LIN {X 0,Y 227.847,Z 291.73,A -85,B 0,C 180,E1 -20016.68,E2 -20016.68} C_VEL
LIN {X 0,Y 227.819,Z 291.734,A -85,B 0,C 180,E1 -20020.379,E2 -20020.379} C_VEL
LIN {X 0,Y 227.828,Z 291.733,A -85,B 0,C 180,E1 -20025.195,E2 -20025.195} C_VEL
LIN {X 0,Y 227.828,Z 291.729,A -85,B 0,C 180,E1 -20029.623,E2 -20029.623} C_VEL
LIN {X 0,Y 227.883,Z 291.723,A -85,B 0,C 180,E1 -20034.128,E2 -20034.128} C_VEL
LIN {X 0,Y 227.87,Z 291.726,A -85,B 0,C 180,E1 -20038.377,E2 -20038.377} C_VEL
LIN {X 0,Y 227.882,Z 291.725,A -85,B 0,C 180,E1 -20042.444,E2 -20042.444} C_VEL
LIN {X 0,Y 227.916,Z 291.719,A -85,B 0,C 180,E1 -20046.368,E2 -20046.368} C_VEL
LIN {X 0,Y 227.945,Z 291.716,A -85,B 0,C 180,E1 -20050.175,E2 -20050.175} C_VEL
LIN {X 0,Y 228.061,Z 291.7,A -85,B 0,C 180,E1 -20053.898,E2 -20053.898} C_VEL
LIN {X 0,Y 228.076,Z 291.698,A -85,B 0,C 180,E1 -20057.543,E2 -20057.543} C_VEL
LIN {X 0,Y 228.26,Z 291.674,A -85,B 0,C 180,E1 -20061.144,E2 -20061.144} C_VEL
LIN {X 0,Y 228.31,Z 291.666,A -85,B 0,C 180,E1 -20062.927,E2 -20062.927} C_VEL
LIN {X 0,Y 228.552,Z 291.64,A -85,B 0,C 180,E1 -20068.238,E2 -20068.238} C_VEL
LIN {X 0,Y 228.554,Z 291.638,A -85,B 0,C 180,E1 -20071.762,E2 -20071.762} C_VEL
LIN {X 0,Y 228.313,Z 291.668,A -85,B 0,C 180,E1 -20077.073,E2 -20077.073} C_VEL
LIN {X 0,Y 228.149,Z 291.687,A -85,B 0,C 180,E1 -20080.651,E2 -20080.651} C_VEL
LIN {X 0,Y 228.068,Z 291.699,A -85,B 0,C 180,E1 -20084.272,E2 -20084.272} C_VEL
LIN {X 0,Y 228.01,Z 291.706,A -85,B 0,C 180,E1 -20087.953,E2 -20087.953} C_VEL
LIN {X 0,Y 227.964,Z 291.712,A -85,B 0,C 180,E1 -20092.348,E2 -20092.348} C_VEL
LIN {X 0,Y 227.945,Z 291.712,A -85,B 0,C 180,E1 -20096.602,E2 -20096.602} C_VEL
LIN {X 0,Y 227.9,Z 291.72,A -85,B 0,C 180,E1 -20100.291,E2 -20100.291} C_VEL
LIN {X 0,Y 227.879,Z 291.72,A -85,B 0,C 180,E1 -20103.72,E2 -20103.72} C_VEL
LIN {X 0,Y 227.842,Z 291.727,A -85,B 0,C 180,E1 -20108.092,E2 -20108.092} C_VEL
LIN {X 0,Y 227.794,Z 291.733,A -85,B 0,C 180,E1 -20112.747,E2 -20112.747} C_VEL
LIN {X 0,Y 227.808,Z 291.733,A -85,B 0,C 180,E1 -20117.256,E2 -20117.256} C_VEL
LIN {X 0,Y 227.847,Z 291.725,A -85,B 0,C 180,E1 -20121.909,E2 -20121.909} C_VEL
LIN {X 0,Y 227.882,Z 291.724,A -85,B 0,C 180,E1 -20126.377,E2 -20126.377} C_VEL
LIN {X 0,Y 227.908,Z 291.719,A -85,B 0,C 180,E1 -20130.436,E2 -20130.436} C_VEL
LIN {X 0,Y 227.932,Z 291.719,A -85,B 0,C 180,E1 -20134.426,E2 -20134.426} C_VEL
LIN {X 0,Y 227.965,Z 291.712,A -85,B 0,C 180,E1 -20138.287,E2 -20138.287} C_VEL
LIN {X 0,Y 228.038,Z 291.703,A -85,B 0,C 180,E1 -20142.825,E2 -20142.825} C_VEL
LIN {X 0,Y 228.076,Z 291.697,A -85,B 0,C 180,E1 -20147.543,E2 -20147.543} C_VEL
LIN {X 0,Y 228.261,Z 291.674,A -85,B 0,C 180,E1 -20151.144,E2 -20151.144} C_VEL
LIN {X 0,Y 228.31,Z 291.666,A -85,B 0,C 180,E1 -20152.927,E2 -20152.927} C_VEL
LIN {X 0,Y 228.554,Z 291.641,A -85,B 0,C 180,E1 -20158.237,E2 -20158.237} C_VEL
LIN {X 0,Y 228.555,Z 291.639,A -85,B 0,C 180,E1 -20161.762,E2 -20161.762} C_VEL
LIN {X 0,Y 228.311,Z 291.669,A -85,B 0,C 180,E1 -20167.072,E2 -20167.072} C_VEL
LIN {X 0,Y 228.148,Z 291.687,A -85,B 0,C 180,E1 -20170.651,E2 -20170.651} C_VEL
LIN {X 0,Y 228.067,Z 291.7,A -85,B 0,C 180,E1 -20174.271,E2 -20174.271} C_VEL
LIN {X 0,Y 228.006,Z 291.706,A -85,B 0,C 180,E1 -20177.953,E2 -20177.953} C_VEL
LIN {X 0,Y 227.925,Z 291.718,A -85,B 0,C 180,E1 -20182.324,E2 -20182.324} C_VEL
LIN {X 0,Y 227.949,Z 291.73,A -85,B 0,C 180,E1 -20185.571,E2 -20185.571} C_VEL
LIN {X 0,Y 228.569,Z 295.999,A -85,B 0,C 180,E1 -20190.577,E2 -20190.577} C_VEL
LIN {X 0,Y 229.068,Z 299.133,A -85,B 0,C 180,E1 -20194.066,E2 -20194.066} C_VEL
LIN {X 0,Y 229.908,Z 303.616,A -85,B 0,C 180,E1 -20198.804,E2 -20198.804} C_VEL
LIN {X 0,Y 230.865,Z 307.87,A -85,B 0,C 180,E1 -20203.062,E2 -20203.062} C_VEL
LIN {X 0,Y 231.268,Z 310.585,A -85,B 0,C 180,E1 -20205.657,E2 -20205.657} C_VEL
LIN {X 0,Y 231.214,Z 313.163,A -85,B 0,C 180,E1 -20208.032,E2 -20208.032} C_VEL
LIN {X 0,Y 230.92,Z 314.73,A -85,B 0,C 180,E1 -20209.433,E2 -20209.433} C_VEL
LIN {X 0,Y 234.651,Z 334.28,A -85,B 0,C 180,E1 -20211.37,E2 -20211.37} C_VEL
LIN {X 0,Y 237.634,Z 350.876,A -85,B 0,C 180,E1 -20213.342,E2 -20213.342} C_VEL
LIN {X 0,Y 240.205,Z 366.69,A -85,B 0,C 180,E1 -20215.507,E2 -20215.507} C_VEL
LIN {X 0,Y 240.445,Z 368.284,A -85,B 0,C 180,E1 -20215.742,E2 -20215.742} C_VEL
LIN {X 0,Y 240.526,Z 373.392,A -85,B 0,C 180,E1 -20216.468,E2 -20216.468} C_VEL
LIN {X 0,Y 239.415,Z 378.527,A -85,B 0,C 180,E1 -20217.164,E2 -20217.164} C_VEL
LIN {X 0,Y 235.584,Z 388.411,A -85,B 0,C 180,E1 -20218.588,E2 -20218.588} C_VEL
LIN {X 0,Y 233.418,Z 394.85,A -85,B 0,C 180,E1 -20219.67,E2 -20219.67} C_VEL
LIN {X 0,Y 230.045,Z 407.856,A -85,B 0,C 180,E1 -20222.281,E2 -20222.281} C_VEL
LIN {X 0,Y 227.246,Z 418.384,A -85,B 0,C 180,E1 -20224.834,E2 -20224.834} C_VEL
LIN {X 0,Y 224.584,Z 429.031,A -85,B 0,C 180,E1 -20227.943,E2 -20227.943} C_VEL
LIN {X 0,Y 222.201,Z 439.134,A -85,B 0,C 180,E1 -20231.561,E2 -20231.561} C_VEL
LIN {X 0,Y 220.517,Z 447.367,A -85,B 0,C 180,E1 -20235.228,E2 -20235.228} C_VEL
LIN {X 0,Y 219.526,Z 453.947,A -85,B 0,C 180,E1 -20238.925,E2 -20238.925} C_VEL
LIN {X 0,Y 219.139,Z 459.038,A -85,B 0,C 180,E1 -20242.629,E2 -20242.629} C_VEL
LIN {X 0,Y 219.1,Z 461.063,A -85,B 0,C 180,E1 -20244.478,E2 -20244.478} C_VEL
LIN {X 0,Y 218.927,Z 464.073,A -85,B 0,C 180,E1 -20248.16,E2 -20248.16} C_VEL
LIN {X 0,Y 218.978,Z 465.12,A -85,B 0,C 180,E1 -20250,E2 -20250} C_VEL
LIN {X 0,Y 218.835,Z 466.296,A -85,B 0,C 180,E1 -20253.683,E2 -20253.683} C_VEL
LIN {X 0,Y 218.754,Z 466.325,A -85,B 0,C 180,E1 -20257.383,E2 -20257.383} C_VEL
LIN {X 0,Y 219.17,Z 465.303,A -85,B 0,C 180,E1 -20261.093,E2 -20261.093} C_VEL
LIN {X 0,Y 220.392,Z 463.369,A -85,B 0,C 180,E1 -20264.78,E2 -20264.78} C_VEL
LIN {X 0,Y 222.497,Z 460.267,A -85,B 0,C 180,E1 -20268.63,E2 -20268.63} C_VEL
LIN {X 0,Y 227.181,Z 454.516,A -85,B 0,C 180,E1 -20273.714,E2 -20273.714} C_VEL
LIN {X 0,Y 232.726,Z 448.077,A -85,B 0,C 180,E1 -20277.91,E2 -20277.91} C_VEL
LIN {X 0,Y 238.908,Z 441.296,A -85,B 0,C 180,E1 -20281.385,E2 -20281.385} C_VEL
LIN {X 0,Y 246.615,Z 433.163,A -85,B 0,C 180,E1 -20284.747,E2 -20284.747} C_VEL
LIN {X 0,Y 256.413,Z 423.002,A -85,B 0,C 180,E1 -20288.076,E2 -20288.076} C_VEL
LIN {X 0,Y 266.397,Z 412.614,A -85,B 0,C 180,E1 -20290.764,E2 -20290.764} C_VEL
LIN {X 0,Y 269.564,Z 409.165,A -85,B 0,C 180,E1 -20291.67,E2 -20291.67} C_VEL
LIN {X 0,Y 273.733,Z 404.367,A -85,B 0,C 180,E1 -20293.189,E2 -20293.189} C_VEL
LIN {X 0,Y 276.225,Z 401.494,A -85,B 0,C 180,E1 -20294.569,E2 -20294.569} C_VEL
LIN {X 0,Y 276.98,Z 400.651,A -85,B 0,C 180,E1 -20295.273,E2 -20295.273} C_VEL
LIN {X 0,Y 276.699,Z 400.883,A -85,B 0,C 180,E1 -20295.995,E2 -20295.995} C_VEL
LIN {X 0,Y 265.948,Z 410.924,A -85,B 0,C 180,E1 -20298.651,E2 -20298.651} C_VEL
LIN {X 0,Y 255.652,Z 420.112,A -85,B 0,C 180,E1 -20301.791,E2 -20301.791} C_VEL
LIN {X 0,Y 246.651,Z 427.81,A -85,B 0,C 180,E1 -20305.259,E2 -20305.259} C_VEL
LIN {X 0,Y 238.941,Z 434.054,A -85,B 0,C 180,E1 -20309.021,E2 -20309.021} C_VEL
LIN {X 0,Y 232.51,Z 438.799,A -85,B 0,C 180,E1 -20313.038,E2 -20313.038} C_VEL
LIN {X 0,Y 228.346,Z 441.537,A -85,B 0,C 180,E1 -20316.415,E2 -20316.415} C_VEL
LIN {X 0,Y 224.998,Z 443.249,A -85,B 0,C 180,E1 -20319.904,E2 -20319.904} C_VEL
LIN {X 0,Y 222.398,Z 443.986,A -85,B 0,C 180,E1 -20323.477,E2 -20323.477} C_VEL
LIN {X 0,Y 220.643,Z 443.701,A -85,B 0,C 180,E1 -20327.117,E2 -20327.117} C_VEL
LIN {X 0,Y 219.572,Z 442.329,A -85,B 0,C 180,E1 -20330.791,E2 -20330.791} C_VEL
LIN {X 0,Y 219.064,Z 439.811,A -85,B 0,C 180,E1 -20334.477,E2 -20334.477} C_VEL
LIN {X 0,Y 218.944,Z 436.124,A -85,B 0,C 180,E1 -20338.161,E2 -20338.161} C_VEL
LIN {X 0,Y 219.045,Z 431.191,A -85,B 0,C 180,E1 -20341.839,E2 -20341.839} C_VEL
LIN {X 0,Y 219.67,Z 424.882,A -85,B 0,C 180,E1 -20345.508,E2 -20345.508} C_VEL
LIN {X 0,Y 220.495,Z 417.013,A -85,B 0,C 180,E1 -20349.171,E2 -20349.171} C_VEL
LIN {X 0,Y 221.966,Z 407.428,A -85,B 0,C 180,E1 -20352.806,E2 -20352.806} C_VEL
LIN {X 0,Y 223.778,Z 397.372,A -85,B 0,C 180,E1 -20355.951,E2 -20355.951} C_VEL
LIN {X 0,Y 226.003,Z 385.408,A -85,B 0,C 180,E1 -20359.058,E2 -20359.058} C_VEL
LIN {X 0,Y 228.56,Z 372.174,A -85,B 0,C 180,E1 -20361.891,E2 -20361.891} C_VEL
LIN {X 0,Y 231.022,Z 358.568,A -85,B 0,C 180,E1 -20364.316,E2 -20364.316} C_VEL
LIN {X 0,Y 233.545,Z 344.768,A -85,B 0,C 180,E1 -20366.351,E2 -20366.351} C_VEL
LIN {X 0,Y 234.092,Z 341.635,A -85,B 0,C 180,E1 -20366.766,E2 -20366.766} C_VEL
LIN {X 0,Y 233.603,Z 337.571,A -85,B 0,C 180,E1 -20367.358,E2 -20367.358} C_VEL
LIN {X 0,Y 230.249,Z 323.156,A -85,B 0,C 180,E1 -20369.415,E2 -20369.415} C_VEL
LIN {X 0,Y 227.217,Z 312.166,A -85,B 0,C 180,E1 -20370.87,E2 -20370.87} C_VEL
LIN {X 0,Y 221.231,Z 294.789,A -85,B 0,C 180,E1 -20373.004,E2 -20373.004} C_VEL
LIN {X 0,Y 220.601,Z 292.633,A -85,B 0,C 180,E1 -20373.269,E2 -20373.269} C_VEL
LIN {X 0,Y 220.793,Z 292.611,A -85,B 0,C 180,E1 -20377.272,E2 -20377.272} C_VEL
LIN {X 0,Y 220.769,Z 292.612,A -85,B 0,C 180,E1 -20381.954,E2 -20381.954} C_VEL
LIN {X 0,Y 220.77,Z 292.61,A -85,B 0,C 180,E1 -20385.545,E2 -20385.545} C_VEL
LIN {X 0,Y 220.809,Z 292.605,A -85,B 0,C 180,E1 -20390.463,E2 -20390.463} C_VEL
LIN {X 0,Y 220.803,Z 292.606,A -85,B 0,C 180,E1 -20395.045,E2 -20395.045} C_VEL
LIN {X 0,Y 220.837,Z 292.6,A -85,B 0,C 180,E1 -20399.39,E2 -20399.39} C_VEL
LIN {X 0,Y 220.897,Z 292.592,A -85,B 0,C 180,E1 -20403.55,E2 -20403.55} C_VEL
LIN {X 0,Y 220.88,Z 292.592,A -85,B 0,C 180,E1 -20407.554,E2 -20407.554} C_VEL
LIN {X 0,Y 220.987,Z 292.582,A -85,B 0,C 180,E1 -20412.571,E2 -20412.571} C_VEL
LIN {X 0,Y 221.015,Z 292.577,A -85,B 0,C 180,E1 -20417.139,E2 -20417.139} C_VEL
LIN {X 0,Y 221.2,Z 292.554,A -85,B 0,C 180,E1 -20420.859,E2 -20420.859} C_VEL
LIN {X 0,Y 221.247,Z 292.546,A -85,B 0,C 180,E1 -20422.7,E2 -20422.7} C_VEL
LIN {X 0,Y 221.509,Z 292.518,A -85,B 0,C 180,E1 -20428.182,E2 -20428.182} C_VEL
LIN {X 0,Y 221.512,Z 292.516,A -85,B 0,C 180,E1 -20431.818,E2 -20431.818} C_VEL
LIN {X 0,Y 221.25,Z 292.549,A -85,B 0,C 180,E1 -20437.3,E2 -20437.3} C_VEL
LIN {X 0,Y 221.07,Z 292.569,A -85,B 0,C 180,E1 -20440.996,E2 -20440.996} C_VEL
LIN {X 0,Y 220.999,Z 292.579,A -85,B 0,C 180,E1 -20444.739,E2 -20444.739} C_VEL
LIN {X 0,Y 220.931,Z 292.586,A -85,B 0,C 180,E1 -20448.549,E2 -20448.549} C_VEL
LIN {X 0,Y 220.924,Z 292.589,A -85,B 0,C 180,E1 -20452.698,E2 -20452.698} C_VEL
LIN {X 0,Y 220.887,Z 292.592,A -85,B 0,C 180,E1 -20457.014,E2 -20457.014} C_VEL
LIN {X 0,Y 220.841,Z 292.6,A -85,B 0,C 180,E1 -20460.768,E2 -20460.768} C_VEL
LIN {X 0,Y 220.796,Z 292.604,A -85,B 0,C 180,E1 -20464.956,E2 -20464.956} C_VEL
LIN {X 0,Y 220.804,Z 292.607,A -85,B 0,C 180,E1 -20467.275,E2 -20467.275} C_VEL
LIN {X 0,Y 220.754,Z 292.607,A -85,B 0,C 180,E1 -20471.957,E2 -20471.957} C_VEL
LIN {X 0,Y 220.768,Z 292.609,A -85,B 0,C 180,E1 -20475.544,E2 -20475.544} C_VEL
LIN {X 0,Y 220.809,Z 292.602,A -85,B 0,C 180,E1 -20480.463,E2 -20480.463} C_VEL
LIN {X 0,Y 220.804,Z 292.606,A -85,B 0,C 180,E1 -20485.045,E2 -20485.045} C_VEL
LIN {X 0,Y 220.837,Z 292.598,A -85,B 0,C 180,E1 -20489.39,E2 -20489.39} C_VEL
LIN {X 0,Y 220.898,Z 292.592,A -85,B 0,C 180,E1 -20493.549,E2 -20493.549} C_VEL
LIN {X 0,Y 220.881,Z 292.591,A -85,B 0,C 180,E1 -20497.553,E2 -20497.553} C_VEL
LIN {X 0,Y 220.988,Z 292.583,A -85,B 0,C 180,E1 -20502.571,E2 -20502.571} C_VEL
LIN {X 0,Y 221.015,Z 292.577,A -85,B 0,C 180,E1 -20507.138,E2 -20507.138} C_VEL
LIN {X 0,Y 221.2,Z 292.554,A -85,B 0,C 180,E1 -20510.859,E2 -20510.859} C_VEL
LIN {X 0,Y 221.126,Z 292.564,A -85,B 0,C 180,E1 -20514.528,E2 -20514.528} C_VEL
LIN {X 0,Y 221.512,Z 292.518,A -85,B 0,C 180,E1 -20518.181,E2 -20518.181} C_VEL
LIN {X 0,Y 221.513,Z 292.516,A -85,B 0,C 180,E1 -20521.818,E2 -20521.818} C_VEL
LIN {X 0,Y 221.248,Z 292.549,A -85,B 0,C 180,E1 -20527.299,E2 -20527.299} C_VEL
LIN {X 0,Y 221.084,Z 292.567,A -85,B 0,C 180,E1 -20530.995,E2 -20530.995} C_VEL
LIN {X 0,Y 221.019,Z 292.576,A -85,B 0,C 180,E1 -20536.629,E2 -20536.629} C_VEL
LIN {X 0,Y 220.891,Z 292.594,A -85,B 0,C 180,E1 -20540.486,E2 -20540.486} C_VEL
LIN {X 0,Y 220.936,Z 292.739,A -85,B 0,C 180,E1 -20545.431,E2 -20545.431} C_VEL
LIN {X 0,Y 221.533,Z 296.956,A -85,B 0,C 180,E1 -20550.503,E2 -20550.503} C_VEL
LIN {X 0,Y 222.115,Z 300.681,A -85,B 0,C 180,E1 -20554.718,E2 -20554.718} C_VEL
LIN {X 0,Y 222.932,Z 304.728,A -85,B 0,C 180,E1 -20559.087,E2 -20559.087} C_VEL
LIN {X 0,Y 223.924,Z 309.32,A -85,B 0,C 180,E1 -20563.79,E2 -20563.79} C_VEL
LIN {X 0,Y 224.233,Z 312.013,A -85,B 0,C 180,E1 -20566.406,E2 -20566.406} C_VEL
LIN {X 0,Y 224.009,Z 314.572,A -85,B 0,C 180,E1 -20568.645,E2 -20568.645} C_VEL
LIN {X 0,Y 227.544,Z 333.061,A -85,B 0,C 180,E1 -20570.548,E2 -20570.548} C_VEL
LIN {X 0,Y 230.371,Z 349.098,A -85,B 0,C 180,E1 -20572.484,E2 -20572.484} C_VEL
LIN {X 0,Y 232.814,Z 364.225,A -85,B 0,C 180,E1 -20574.592,E2 -20574.592} C_VEL
LIN {X 0,Y 235.019,Z 379.599,A -85,B 0,C 180,E1 -20577.052,E2 -20577.052} C_VEL
LIN {X 0,Y 235.709,Z 385.312,A -85,B 0,C 180,E1 -20578.045,E2 -20578.045} C_VEL
LIN {X 0,Y 233.418,Z 394.85,A -85,B 0,C 180,E1 -20579.67,E2 -20579.67} C_VEL
LIN {X 0,Y 231.667,Z 399.404,A -85,B 0,C 180,E1 -20580.493,E2 -20580.493} C_VEL
LIN {X 0,Y 227.025,Z 406.366,A -85,B 0,C 180,E1 -20581.819,E2 -20581.819} C_VEL
LIN {X 0,Y 222.322,Z 413.006,A -85,B 0,C 180,E1 -20583.286,E2 -20583.286} C_VEL
LIN {X 0,Y 220.509,Z 417.005,A -85,B 0,C 180,E1 -20584.315,E2 -20584.315} C_VEL
LIN {X 0,Y 217.61,Z 428.329,A -85,B 0,C 180,E1 -20587.698,E2 -20587.698} C_VEL
LIN {X 0,Y 215.295,Z 437.86,A -85,B 0,C 180,E1 -20591.201,E2 -20591.201} C_VEL
LIN {X 0,Y 213.635,Z 445.704,A -85,B 0,C 180,E1 -20594.741,E2 -20594.741} C_VEL
LIN {X 0,Y 212.564,Z 452.501,A -85,B 0,C 180,E1 -20598.558,E2 -20598.558} C_VEL
LIN {X 0,Y 212.131,Z 457.789,A -85,B 0,C 180,E1 -20602.385,E2 -20602.385} C_VEL
LIN {X 0,Y 212.067,Z 459.908,A -85,B 0,C 180,E1 -20604.294,E2 -20604.294} C_VEL
LIN {X 0,Y 211.895,Z 463.117,A -85,B 0,C 180,E1 -20608.099,E2 -20608.099} C_VEL
LIN {X 0,Y 211.936,Z 464.26,A -85,B 0,C 180,E1 -20610,E2 -20610} C_VEL
LIN {X 0,Y 211.771,Z 465.581,A -85,B 0,C 180,E1 -20613.806,E2 -20613.806} C_VEL
LIN {X 0,Y 211.68,Z 465.763,A -85,B 0,C 180,E1 -20617.632,E2 -20617.632} C_VEL
LIN {X 0,Y 212.163,Z 464.983,A -85,B 0,C 180,E1 -20621.464,E2 -20621.464} C_VEL
LIN {X 0,Y 213.485,Z 463.196,A -85,B 0,C 180,E1 -20625.27,E2 -20625.27} C_VEL
LIN {X 0,Y 215.588,Z 460.565,A -85,B 0,C 180,E1 -20629.026,E2 -20629.026} C_VEL
LIN {X 0,Y 219.701,Z 456.074,A -85,B 0,C 180,E1 -20633.57,E2 -20633.57} C_VEL
LIN {X 0,Y 225.199,Z 450.318,A -85,B 0,C 180,E1 -20637.912,E2 -20637.912} C_VEL
LIN {X 0,Y 232.09,Z 443.521,A -85,B 0,C 180,E1 -20641.84,E2 -20641.84} C_VEL
LIN {X 0,Y 241.018,Z 435.027,A -85,B 0,C 180,E1 -20645.676,E2 -20645.676} C_VEL
LIN {X 0,Y 250.062,Z 426.505,A -85,B 0,C 180,E1 -20648.707,E2 -20648.707} C_VEL
LIN {X 0,Y 260.195,Z 416.935,A -85,B 0,C 180,E1 -20651.434,E2 -20651.434} C_VEL
LIN {X 0,Y 264.861,Z 412.456,A -85,B 0,C 180,E1 -20652.582,E2 -20652.582} C_VEL
LIN {X 0,Y 268.699,Z 408.536,A -85,B 0,C 180,E1 -20653.851,E2 -20653.851} C_VEL
LIN {X 0,Y 270.34,Z 406.877,A -85,B 0,C 180,E1 -20654.581,E2 -20654.581} C_VEL
LIN {X 0,Y 270.594,Z 406.481,A -85,B 0,C 180,E1 -20655.472,E2 -20655.472} C_VEL
LIN {X 0,Y 258.984,Z 416.184,A -85,B 0,C 180,E1 -20658.329,E2 -20658.329} C_VEL
LIN {X 0,Y 248.57,Z 424.466,A -85,B 0,C 180,E1 -20661.536,E2 -20661.536} C_VEL
LIN {X 0,Y 239.441,Z 431.354,A -85,B 0,C 180,E1 -20665.086,E2 -20665.086} C_VEL
LIN {X 0,Y 231.611,Z 436.866,A -85,B 0,C 180,E1 -20668.946,E2 -20668.946} C_VEL
LIN {X 0,Y 226.327,Z 440.227,A -85,B 0,C 180,E1 -20672.239,E2 -20672.239} C_VEL
LIN {X 0,Y 221.905,Z 442.671,A -85,B 0,C 180,E1 -20675.687,E2 -20675.687} C_VEL
LIN {X 0,Y 218.362,Z 444.198,A -85,B 0,C 180,E1 -20679.266,E2 -20679.266} C_VEL
LIN {X 0,Y 215.596,Z 444.699,A -85,B 0,C 180,E1 -20682.94,E2 -20682.94} C_VEL
LIN {X 0,Y 213.695,Z 444.182,A -85,B 0,C 180,E1 -20686.691,E2 -20686.691} C_VEL
LIN {X 0,Y 212.538,Z 442.621,A -85,B 0,C 180,E1 -20690.484,E2 -20690.484} C_VEL
LIN {X 0,Y 211.981,Z 439.964,A -85,B 0,C 180,E1 -20694.292,E2 -20694.292} C_VEL
LIN {X 0,Y 211.852,Z 436.119,A -85,B 0,C 180,E1 -20698.099,E2 -20698.099} C_VEL
LIN {X 0,Y 211.978,Z 430.991,A -85,B 0,C 180,E1 -20701.9,E2 -20701.9} C_VEL
LIN {X 0,Y 212.615,Z 424.513,A -85,B 0,C 180,E1 -20705.692,E2 -20705.692} C_VEL
LIN {X 0,Y 213.498,Z 416.474,A -85,B 0,C 180,E1 -20709.474,E2 -20709.474} C_VEL
LIN {X 0,Y 215.023,Z 406.652,A -85,B 0,C 180,E1 -20713.227,E2 -20713.227} C_VEL
LIN {X 0,Y 216.929,Z 396.37,A -85,B 0,C 180,E1 -20716.468,E2 -20716.468} C_VEL
LIN {X 0,Y 219.272,Z 384.17,A -85,B 0,C 180,E1 -20719.667,E2 -20719.667} C_VEL
LIN {X 0,Y 221.719,Z 371.799,A -85,B 0,C 180,E1 -20722.357,E2 -20722.357} C_VEL
LIN {X 0,Y 224.191,Z 358.428,A -85,B 0,C 180,E1 -20724.789,E2 -20724.789} C_VEL
LIN {X 0,Y 226.869,Z 344.085,A -85,B 0,C 180,E1 -20726.94,E2 -20726.94} C_VEL
LIN {X 0,Y 227.131,Z 340.848,A -85,B 0,C 180,E1 -20727.405,E2 -20727.405} C_VEL
LIN {X 0,Y 223.608,Z 325.306,A -85,B 0,C 180,E1 -20729.744,E2 -20729.744} C_VEL
LIN {X 0,Y 220.552,Z 314.174,A -85,B 0,C 180,E1 -20731.293,E2 -20731.293} C_VEL
LIN {X 0,Y 215.65,Z 299.656,A -85,B 0,C 180,E1 -20733.19,E2 -20733.19} C_VEL
LIN {X 0,Y 213.59,Z 293.503,A -85,B 0,C 180,E1 -20733.943,E2 -20733.943} C_VEL
LIN {X 0,Y 213.713,Z 293.491,A -85,B 0,C 180,E1 -20737.885,E2 -20737.885} C_VEL
LIN {X 0,Y 213.71,Z 293.493,A -85,B 0,C 180,E1 -20741.126,E2 -20741.126} C_VEL
LIN {X 0,Y 213.705,Z 293.491,A -85,B 0,C 180,E1 -20743.68,E2 -20743.68} C_VEL
LIN {X 0,Y 213.705,Z 293.491,A -85,B 0,C 180,E1 -20746.345,E2 -20746.345} C_VEL
LIN {X 0,Y 213.719,Z 293.489,A -85,B 0,C 180,E1 -20749.143,E2 -20749.143} C_VEL
LIN {X 0,Y 213.746,Z 293.483,A -85,B 0,C 180,E1 -20753.712,E2 -20753.712} C_VEL
LIN {X 0,Y 213.783,Z 293.481,A -85,B 0,C 180,E1 -20758.732,E2 -20758.732} C_VEL
LIN {X 0,Y 213.829,Z 293.476,A -85,B 0,C 180,E1 -20762.603,E2 -20762.603} C_VEL
LIN {X 0,Y 213.855,Z 293.468,A -85,B 0,C 180,E1 -20766.953,E2 -20766.953} C_VEL
LIN {X 0,Y 213.947,Z 293.458,A -85,B 0,C 180,E1 -20772.804,E2 -20772.804} C_VEL
LIN {X 0,Y 213.957,Z 293.457,A -85,B 0,C 180,E1 -20776.707,E2 -20776.707} C_VEL
LIN {X 0,Y 214.139,Z 293.435,A -85,B 0,C 180,E1 -20780.555,E2 -20780.555} C_VEL
LIN {X 0,Y 214.085,Z 293.442,A -85,B 0,C 180,E1 -20784.348,E2 -20784.348} C_VEL
LIN {X 0,Y 214.442,Z 293.399,A -85,B 0,C 180,E1 -20788.122,E2 -20788.122} C_VEL
LIN {X 0,Y 214.545,Z 293.384,A -85,B 0,C 180,E1 -20790,E2 -20790} C_VEL
LIN {X 0,Y 214.445,Z 293.396,A -85,B 0,C 180,E1 -20791.878,E2 -20791.878} C_VEL
LIN {X 0,Y 214.191,Z 293.429,A -85,B 0,C 180,E1 -20797.542,E2 -20797.542} C_VEL
LIN {X 0,Y 214.002,Z 293.451,A -85,B 0,C 180,E1 -20801.364,E2 -20801.364} C_VEL
LIN {X 0,Y 213.937,Z 293.461,A -85,B 0,C 180,E1 -20805.237,E2 -20805.237} C_VEL
LIN {X 0,Y 213.88,Z 293.466,A -85,B 0,C 180,E1 -20809.184,E2 -20809.184} C_VEL
LIN {X 0,Y 213.859,Z 293.471,A -85,B 0,C 180,E1 -20813.226,E2 -20813.226} C_VEL
LIN {X 0,Y 213.832,Z 293.474,A -85,B 0,C 180,E1 -20817.45,E2 -20817.45} C_VEL
LIN {X 0,Y 213.77,Z 293.48,A -85,B 0,C 180,E1 -20821.737,E2 -20821.737} C_VEL
LIN {X 0,Y 213.744,Z 293.482,A -85,B 0,C 180,E1 -20826.289,E2 -20826.289} C_VEL
LIN {X 0,Y 213.702,Z 293.489,A -85,B 0,C 180,E1 -20831.128,E2 -20831.128} C_VEL
LIN {X 0,Y 213.704,Z 293.487,A -85,B 0,C 180,E1 -20833.679,E2 -20833.679} C_VEL
LIN {X 0,Y 213.705,Z 293.489,A -85,B 0,C 180,E1 -20836.345,E2 -20836.345} C_VEL
LIN {X 0,Y 213.719,Z 293.486,A -85,B 0,C 180,E1 -20839.143,E2 -20839.143} C_VEL
LIN {X 0,Y 213.747,Z 293.483,A -85,B 0,C 180,E1 -20843.712,E2 -20843.712} C_VEL
LIN {X 0,Y 213.783,Z 293.478,A -85,B 0,C 180,E1 -20848.731,E2 -20848.731} C_VEL
LIN {X 0,Y 213.829,Z 293.476,A -85,B 0,C 180,E1 -20852.603,E2 -20852.603} C_VEL
LIN {X 0,Y 213.855,Z 293.467,A -85,B 0,C 180,E1 -20856.953,E2 -20856.953} C_VEL
LIN {X 0,Y 213.947,Z 293.458,A -85,B 0,C 180,E1 -20862.803,E2 -20862.803} C_VEL
LIN {X 0,Y 213.957,Z 293.457,A -85,B 0,C 180,E1 -20866.706,E2 -20866.706} C_VEL
LIN {X 0,Y 214.139,Z 293.435,A -85,B 0,C 180,E1 -20870.555,E2 -20870.555} C_VEL
LIN {X 0,Y 214.088,Z 293.441,A -85,B 0,C 180,E1 -20874.348,E2 -20874.348} C_VEL
LIN {X 0,Y 214.444,Z 293.399,A -85,B 0,C 180,E1 -20878.121,E2 -20878.121} C_VEL
LIN {X 0,Y 214.542,Z 293.386,A -85,B 0,C 180,E1 -20880,E2 -20880} C_VEL
LIN {X 0,Y 214.446,Z 293.396,A -85,B 0,C 180,E1 -20881.878,E2 -20881.878} C_VEL
LIN {X 0,Y 214.189,Z 293.43,A -85,B 0,C 180,E1 -20887.541,E2 -20887.541} C_VEL
LIN {X 0,Y 214.01,Z 293.449,A -85,B 0,C 180,E1 -20891.363,E2 -20891.363} C_VEL
LIN {X 0,Y 213.937,Z 293.461,A -85,B 0,C 180,E1 -20895.236,E2 -20895.236} C_VEL
LIN {X 0,Y 213.84,Z 293.47,A -85,B 0,C 180,E1 -20899.187,E2 -20899.187} C_VEL
LIN {X 0,Y 213.859,Z 293.472,A -85,B 0,C 180,E1 -20904.771,E2 -20904.771} C_VEL
LIN {X 0,Y 214.339,Z 297.088,A -85,B 0,C 180,E1 -20909.461,E2 -20909.461} C_VEL
LIN {X 0,Y 214.914,Z 300.757,A -85,B 0,C 180,E1 -20913.774,E2 -20913.774} C_VEL
LIN {X 0,Y 215.773,Z 305.06,A -85,B 0,C 180,E1 -20918.582,E2 -20918.582} C_VEL
LIN {X 0,Y 216.695,Z 309.15,A -85,B 0,C 180,E1 -20922.928,E2 -20922.928} C_VEL
LIN {X 0,Y 217.068,Z 311.606,A -85,B 0,C 180,E1 -20925.421,E2 -20925.421} C_VEL
LIN {X 0,Y 217.052,Z 314.034,A -85,B 0,C 180,E1 -20927.794,E2 -20927.794} C_VEL
LIN {X 0,Y 220.685,Z 333.154,A -85,B 0,C 180,E1 -20929.845,E2 -20929.845} C_VEL
LIN {X 0,Y 223.594,Z 350.185,A -85,B 0,C 180,E1 -20931.994,E2 -20931.994} C_VEL
LIN {X 0,Y 226.018,Z 365.905,A -85,B 0,C 180,E1 -20934.301,E2 -20934.301} C_VEL
LIN {X 0,Y 228.129,Z 381.104,A -85,B 0,C 180,E1 -20936.85,E2 -20936.85} C_VEL
LIN {X 0,Y 228.709,Z 385.93,A -85,B 0,C 180,E1 -20937.729,E2 -20937.729} C_VEL
LIN {X 0,Y 225.445,Z 398.804,A -85,B 0,C 180,E1 -20940.08,E2 -20940.08} C_VEL
LIN {X 0,Y 222.174,Z 410.971,A -85,B 0,C 180,E1 -20942.77,E2 -20942.77} C_VEL
LIN {X 0,Y 220.509,Z 417.005,A -85,B 0,C 180,E1 -20944.315,E2 -20944.315} C_VEL
LIN {X 0,Y 218.76,Z 420.912,A -85,B 0,C 180,E1 -20945.386,E2 -20945.386} C_VEL
LIN {X 0,Y 214.35,Z 426.752,A -85,B 0,C 180,E1 -20947.155,E2 -20947.155} C_VEL
LIN {X 0,Y 210.101,Z 432.21,A -85,B 0,C 180,E1 -20949.082,E2 -20949.082} C_VEL
LIN {X 0,Y 208.638,Z 435.459,A -85,B 0,C 180,E1 -20950.377,E2 -20950.377} C_VEL
LIN {X 0,Y 206.773,Z 443.988,A -85,B 0,C 180,E1 -20954.222,E2 -20954.222} C_VEL
LIN {X 0,Y 205.616,Z 450.999,A -85,B 0,C 180,E1 -20958.166,E2 -20958.166} C_VEL
LIN {X 0,Y 205.102,Z 456.499,A -85,B 0,C 180,E1 -20962.122,E2 -20962.122} C_VEL
LIN {X 0,Y 205.033,Z 458.72,A -85,B 0,C 180,E1 -20964.098,E2 -20964.098} C_VEL
LIN {X 0,Y 204.862,Z 462.12,A -85,B 0,C 180,E1 -20968.034,E2 -20968.034} C_VEL
LIN {X 0,Y 204.915,Z 463.321,A -85,B 0,C 180,E1 -20970,E2 -20970} C_VEL
LIN {X 0,Y 204.707,Z 464.793,A -85,B 0,C 180,E1 -20973.937,E2 -20973.937} C_VEL
LIN {X 0,Y 204.613,Z 465.196,A -85,B 0,C 180,E1 -20977.897,E2 -20977.897} C_VEL
LIN {X 0,Y 205.153,Z 464.562,A -85,B 0,C 180,E1 -20981.861,E2 -20981.861} C_VEL
LIN {X 0,Y 206.567,Z 463.031,A -85,B 0,C 180,E1 -20985.794,E2 -20985.794} C_VEL
LIN {X 0,Y 208.848,Z 460.625,A -85,B 0,C 180,E1 -20989.665,E2 -20989.665} C_VEL
LIN {X 0,Y 214.235,Z 455.519,A -85,B 0,C 180,E1 -20995.244,E2 -20995.244} C_VEL
LIN {X 0,Y 220.359,Z 449.901,A -85,B 0,C 180,E1 -20999.627,E2 -20999.627} C_VEL
LIN {X 0,Y 228.165,Z 443.095,A -85,B 0,C 180,E1 -21003.672,E2 -21003.672} C_VEL
LIN {X 0,Y 237.439,Z 435.139,A -85,B 0,C 180,E1 -21007.358,E2 -21007.358} C_VEL
LIN {X 0,Y 248.199,Z 426,A -85,B 0,C 180,E1 -21010.638,E2 -21010.638} C_VEL
LIN {X 0,Y 260.18,Z 415.651,A -85,B 0,C 180,E1 -21013.536,E2 -21013.536} C_VEL
LIN {X 0,Y 263.973,Z 412.244,A -85,B 0,C 180,E1 -21014.689,E2 -21014.689} C_VEL
LIN {X 0,Y 263.176,Z 412.766,A -85,B 0,C 180,E1 -21015.195,E2 -21015.195} C_VEL
LIN {X 0,Y 252.001,Z 421.096,A -85,B 0,C 180,E1 -21017.985,E2 -21017.985} C_VEL
LIN {X 0,Y 243.455,Z 427.182,A -85,B 0,C 180,E1 -21020.574,E2 -21020.574} C_VEL
LIN {X 0,Y 233.125,Z 434.05,A -85,B 0,C 180,E1 -21024.486,E2 -21024.486} C_VEL
LIN {X 0,Y 225.746,Z 438.586,A -85,B 0,C 180,E1 -21028.046,E2 -21028.046} C_VEL
LIN {X 0,Y 220.188,Z 441.676,A -85,B 0,C 180,E1 -21031.395,E2 -21031.395} C_VEL
LIN {X 0,Y 215.51,Z 443.825,A -85,B 0,C 180,E1 -21034.917,E2 -21034.917} C_VEL
LIN {X 0,Y 211.727,Z 445.074,A -85,B 0,C 180,E1 -21038.585,E2 -21038.585} C_VEL
LIN {X 0,Y 208.818,Z 445.393,A -85,B 0,C 180,E1 -21042.368,E2 -21042.368} C_VEL
LIN {X 0,Y 206.766,Z 444.653,A -85,B 0,C 180,E1 -21046.236,E2 -21046.236} C_VEL
LIN {X 0,Y 205.508,Z 442.874,A -85,B 0,C 180,E1 -21050.155,E2 -21050.155} C_VEL
LIN {X 0,Y 204.901,Z 440.03,A -85,B 0,C 180,E1 -21054.094,E2 -21054.094} C_VEL
LIN {X 0,Y 204.763,Z 436.017,A -85,B 0,C 180,E1 -21058.034,E2 -21058.034} C_VEL
LIN {X 0,Y 204.913,Z 430.769,A -85,B 0,C 180,E1 -21061.966,E2 -21061.966} C_VEL
LIN {X 0,Y 205.561,Z 424.079,A -85,B 0,C 180,E1 -21065.888,E2 -21065.888} C_VEL
LIN {X 0,Y 206.496,Z 415.822,A -85,B 0,C 180,E1 -21069.798,E2 -21069.798} C_VEL
LIN {X 0,Y 208.088,Z 405.779,A -85,B 0,C 180,E1 -21073.676,E2 -21073.676} C_VEL
LIN {X 0,Y 210.106,Z 395.244,A -85,B 0,C 180,E1 -21077.019,E2 -21077.019} C_VEL
LIN {X 0,Y 212.566,Z 382.756,A -85,B 0,C 180,E1 -21080.314,E2 -21080.314} C_VEL
LIN {X 0,Y 214.893,Z 371.268,A -85,B 0,C 180,E1 -21082.854,E2 -21082.854} C_VEL
LIN {X 0,Y 217.715,Z 356.547,A -85,B 0,C 180,E1 -21085.579,E2 -21085.579} C_VEL
LIN {X 0,Y 220.212,Z 343.409,A -85,B 0,C 180,E1 -21087.566,E2 -21087.566} C_VEL
LIN {X 0,Y 219.749,Z 339.789,A -85,B 0,C 180,E1 -21088.147,E2 -21088.147} C_VEL
LIN {X 0,Y 216.654,Z 326.188,A -85,B 0,C 180,E1 -21090.267,E2 -21090.267} C_VEL
LIN {X 0,Y 213.851,Z 316.062,A -85,B 0,C 180,E1 -21091.724,E2 -21091.724} C_VEL
LIN {X 0,Y 208.588,Z 300.478,A -85,B 0,C 180,E1 -21093.855,E2 -21093.855} C_VEL
LIN {X 0,Y 206.573,Z 294.388,A -85,B 0,C 180,E1 -21094.613,E2 -21094.613} C_VEL
LIN {X 0,Y 206.672,Z 294.369,A -85,B 0,C 180,E1 -21098.544,E2 -21098.544} C_VEL
LIN {X 0,Y 206.624,Z 294.377,A -85,B 0,C 180,E1 -21102.866,E2 -21102.866} C_VEL
LIN {X 0,Y 206.625,Z 294.372,A -85,B 0,C 180,E1 -21107.135,E2 -21107.135} C_VEL
LIN {X 0,Y 206.69,Z 294.363,A -85,B 0,C 180,E1 -21111.45,E2 -21111.45} C_VEL
LIN {X 0,Y 206.702,Z 294.364,A -85,B 0,C 180,E1 -21114.689,E2 -21114.689} C_VEL
LIN {X 0,Y 206.709,Z 294.36,A -85,B 0,C 180,E1 -21119.337,E2 -21119.337} C_VEL
LIN {X 0,Y 206.735,Z 294.356,A -85,B 0,C 180,E1 -21123.772,E2 -21123.772} C_VEL
LIN {X 0,Y 206.76,Z 294.352,A -85,B 0,C 180,E1 -21128.043,E2 -21128.043} C_VEL
LIN {X 0,Y 206.877,Z 294.341,A -85,B 0,C 180,E1 -21132.197,E2 -21132.197} C_VEL
LIN {X 0,Y 206.899,Z 294.337,A -85,B 0,C 180,E1 -21136.245,E2 -21136.245} C_VEL
LIN {X 0,Y 207.083,Z 294.315,A -85,B 0,C 180,E1 -21140.23,E2 -21140.23} C_VEL
LIN {X 0,Y 207.047,Z 294.318,A -85,B 0,C 180,E1 -21144.155,E2 -21144.155} C_VEL
LIN {X 0,Y 207.378,Z 294.279,A -85,B 0,C 180,E1 -21148.058,E2 -21148.058} C_VEL
LIN {X 0,Y 207.511,Z 294.26,A -85,B 0,C 180,E1 -21150,E2 -21150} C_VEL
LIN {X 0,Y 207.381,Z 294.276,A -85,B 0,C 180,E1 -21151.942,E2 -21151.942} C_VEL
LIN {X 0,Y 207.135,Z 294.308,A -85,B 0,C 180,E1 -21157.8,E2 -21157.8} C_VEL
LIN {X 0,Y 206.928,Z 294.335,A -85,B 0,C 180,E1 -21161.758,E2 -21161.758} C_VEL
LIN {X 0,Y 206.871,Z 294.34,A -85,B 0,C 180,E1 -21165.771,E2 -21165.771} C_VEL
LIN {X 0,Y 206.816,Z 294.348,A -85,B 0,C 180,E1 -21169.866,E2 -21169.866} C_VEL
LIN {X 0,Y 206.771,Z 294.351,A -85,B 0,C 180,E1 -21174.071,E2 -21174.071} C_VEL
LIN {X 0,Y 206.74,Z 294.355,A -85,B 0,C 180,E1 -21178.42,E2 -21178.42} C_VEL
LIN {X 0,Y 206.701,Z 294.362,A -85,B 0,C 180,E1 -21182.958,E2 -21182.958} C_VEL
LIN {X 0,Y 206.671,Z 294.365,A -85,B 0,C 180,E1 -21187.742,E2 -21187.742} C_VEL
LIN {X 0,Y 206.635,Z 294.367,A -85,B 0,C 180,E1 -21191.559,E2 -21191.559} C_VEL
LIN {X 0,Y 206.633,Z 294.37,A -85,B 0,C 180,E1 -21195.582,E2 -21195.582} C_VEL
LIN {X 0,Y 206.663,Z 294.363,A -85,B 0,C 180,E1 -21199.749,E2 -21199.749} C_VEL
LIN {X 0,Y 206.702,Z 294.363,A -85,B 0,C 180,E1 -21204.689,E2 -21204.689} C_VEL
LIN {X 0,Y 206.71,Z 294.357,A -85,B 0,C 180,E1 -21209.336,E2 -21209.336} C_VEL
LIN {X 0,Y 206.736,Z 294.357,A -85,B 0,C 180,E1 -21213.772,E2 -21213.772} C_VEL
LIN {X 0,Y 206.761,Z 294.351,A -85,B 0,C 180,E1 -21218.043,E2 -21218.043} C_VEL
LIN {X 0,Y 206.877,Z 294.341,A -85,B 0,C 180,E1 -21222.196,E2 -21222.196} C_VEL
LIN {X 0,Y 206.899,Z 294.335,A -85,B 0,C 180,E1 -21226.244,E2 -21226.244} C_VEL
LIN {X 0,Y 207.083,Z 294.316,A -85,B 0,C 180,E1 -21230.23,E2 -21230.23} C_VEL
LIN {X 0,Y 207.05,Z 294.317,A -85,B 0,C 180,E1 -21234.155,E2 -21234.155} C_VEL
LIN {X 0,Y 207.381,Z 294.279,A -85,B 0,C 180,E1 -21238.057,E2 -21238.057} C_VEL
LIN {X 0,Y 207.508,Z 294.262,A -85,B 0,C 180,E1 -21240,E2 -21240} C_VEL
LIN {X 0,Y 207.383,Z 294.275,A -85,B 0,C 180,E1 -21241.942,E2 -21241.942} C_VEL
LIN {X 0,Y 207.133,Z 294.309,A -85,B 0,C 180,E1 -21247.8,E2 -21247.8} C_VEL
LIN {X 0,Y 206.934,Z 294.333,A -85,B 0,C 180,E1 -21251.757,E2 -21251.757} C_VEL
LIN {X 0,Y 206.87,Z 294.341,A -85,B 0,C 180,E1 -21255.77,E2 -21255.77} C_VEL
LIN {X 0,Y 206.783,Z 294.353,A -85,B 0,C 180,E1 -21259.869,E2 -21259.869} C_VEL
LIN {X 0,Y 206.831,Z 294.465,A -85,B 0,C 180,E1 -21264.865,E2 -21264.865} C_VEL
LIN {X 0,Y 207.163,Z 297.191,A -85,B 0,C 180,E1 -21268.356,E2 -21268.356} C_VEL
LIN {X 0,Y 207.722,Z 300.806,A -85,B 0,C 180,E1 -21272.774,E2 -21272.774} C_VEL
LIN {X 0,Y 208.47,Z 304.75,A -85,B 0,C 180,E1 -21277.359,E2 -21277.359} C_VEL
LIN {X 0,Y 209.504,Z 309.352,A -85,B 0,C 180,E1 -21282.437,E2 -21282.437} C_VEL
LIN {X 0,Y 209.983,Z 312.106,A -85,B 0,C 180,E1 -21285.343,E2 -21285.343} C_VEL
LIN {X 0,Y 209.998,Z 313.659,A -85,B 0,C 180,E1 -21286.921,E2 -21286.921} C_VEL
LIN {X 0,Y 213.444,Z 331.306,A -85,B 0,C 180,E1 -21288.892,E2 -21288.892} C_VEL
LIN {X 0,Y 216.156,Z 347.138,A -85,B 0,C 180,E1 -21290.927,E2 -21290.927} C_VEL
LIN {X 0,Y 218.591,Z 362.965,A -85,B 0,C 180,E1 -21293.266,E2 -21293.266} C_VEL
LIN {X 0,Y 220.696,Z 378.433,A -85,B 0,C 180,E1 -21295.889,E2 -21295.889} C_VEL
LIN {X 0,Y 221.684,Z 386.352,A -85,B 0,C 180,E1 -21297.388,E2 -21297.388} C_VEL
LIN {X 0,Y 218.059,Z 400.104,A -85,B 0,C 180,E1 -21300.029,E2 -21300.029} C_VEL
LIN {X 0,Y 214.904,Z 411.718,A -85,B 0,C 180,E1 -21302.752,E2 -21302.752} C_VEL
LIN {X 0,Y 211.752,Z 423.183,A -85,B 0,C 180,E1 -21306.01,E2 -21306.01} C_VEL
LIN {X 0,Y 209.269,Z 432.838,A -85,B 0,C 180,E1 -21309.352,E2 -21309.352} C_VEL
LIN {X 0,Y 208.638,Z 435.459,A -85,B 0,C 180,E1 -21310.377,E2 -21310.377} C_VEL
LIN {X 0,Y 207.245,Z 438.604,A -85,B 0,C 180,E1 -21311.709,E2 -21311.709} C_VEL
LIN {X 0,Y 203.395,Z 443.11,A -85,B 0,C 180,E1 -21313.922,E2 -21313.922} C_VEL
LIN {X 0,Y 199.733,Z 447.187,A -85,B 0,C 180,E1 -21316.285,E2 -21316.285} C_VEL
LIN {X 0,Y 198.665,Z 449.551,A -85,B 0,C 180,E1 -21317.821,E2 -21317.821} C_VEL
LIN {X 0,Y 198.093,Z 455.135,A -85,B 0,C 180,E1 -21321.841,E2 -21321.841} C_VEL
LIN {X 0,Y 198.037,Z 457.441,A -85,B 0,C 180,E1 -21323.888,E2 -21323.888} C_VEL
LIN {X 0,Y 197.852,Z 461,A -85,B 0,C 180,E1 -21327.964,E2 -21327.964} C_VEL
LIN {X 0,Y 197.893,Z 462.305,A -85,B 0,C 180,E1 -21330,E2 -21330} C_VEL
LIN {X 0,Y 197.647,Z 463.989,A -85,B 0,C 180,E1 -21334.078,E2 -21334.078} C_VEL
LIN {X 0,Y 197.567,Z 464.535,A -85,B 0,C 180,E1 -21338.18,E2 -21338.18} C_VEL
LIN {X 0,Y 198.163,Z 464.122,A -85,B 0,C 180,E1 -21342.286,E2 -21342.286} C_VEL
LIN {X 0,Y 199.671,Z 462.814,A -85,B 0,C 180,E1 -21346.355,E2 -21346.355} C_VEL
LIN {X 0,Y 202.127,Z 460.648,A -85,B 0,C 180,E1 -21350.347,E2 -21350.347} C_VEL
LIN {X 0,Y 205.679,Z 457.703,A -85,B 0,C 180,E1 -21354.207,E2 -21354.207} C_VEL
LIN {X 0,Y 212.807,Z 451.906,A -85,B 0,C 180,E1 -21359.695,E2 -21359.695} C_VEL
LIN {X 0,Y 218.936,Z 447.092,A -85,B 0,C 180,E1 -21363.073,E2 -21363.073} C_VEL
LIN {X 0,Y 228.002,Z 440.134,A -85,B 0,C 180,E1 -21366.947,E2 -21366.947} C_VEL
LIN {X 0,Y 238.526,Z 432.084,A -85,B 0,C 180,E1 -21370.407,E2 -21370.407} C_VEL
LIN {X 0,Y 250.372,Z 422.862,A -85,B 0,C 180,E1 -21373.45,E2 -21373.45} C_VEL
LIN {X 0,Y 255.692,Z 418.656,A -85,B 0,C 180,E1 -21374.594,E2 -21374.594} C_VEL
LIN {X 0,Y 255.228,Z 418.897,A -85,B 0,C 180,E1 -21375.015,E2 -21375.015} C_VEL
LIN {X 0,Y 242.718,Z 427.119,A -85,B 0,C 180,E1 -21378.243,E2 -21378.243} C_VEL
LIN {X 0,Y 232.326,Z 433.487,A -85,B 0,C 180,E1 -21381.674,E2 -21381.674} C_VEL
LIN {X 0,Y 223.207,Z 438.626,A -85,B 0,C 180,E1 -21385.476,E2 -21385.476} C_VEL
LIN {X 0,Y 216.916,Z 441.77,A -85,B 0,C 180,E1 -21388.776,E2 -21388.776} C_VEL
LIN {X 0,Y 211.55,Z 444.105,A -85,B 0,C 180,E1 -21392.284,E2 -21392.284} C_VEL
LIN {X 0,Y 207.067,Z 445.57,A -85,B 0,C 180,E1 -21395.966,E2 -21395.966} C_VEL
LIN {X 0,Y 203.507,Z 446.081,A -85,B 0,C 180,E1 -21399.798,E2 -21399.798} C_VEL
LIN {X 0,Y 200.78,Z 445.669,A -85,B 0,C 180,E1 -21403.739,E2 -21403.739} C_VEL
LIN {X 0,Y 199.071,Z 444.236,A -85,B 0,C 180,E1 -21407.771,E2 -21407.771} C_VEL
LIN {X 0,Y 198.077,Z 441.713,A -85,B 0,C 180,E1 -21411.841,E2 -21411.841} C_VEL
LIN {X 0,Y 197.678,Z 438.101,A -85,B 0,C 180,E1 -21415.923,E2 -21415.923} C_VEL
LIN {X 0,Y 197.738,Z 433.287,A -85,B 0,C 180,E1 -21420,E2 -21420} C_VEL
LIN {X 0,Y 198.143,Z 427.15,A -85,B 0,C 180,E1 -21424.068,E2 -21424.068} C_VEL
LIN {X 0,Y 198.764,Z 420.619,A -85,B 0,C 180,E1 -21427.605,E2 -21427.605} C_VEL
LIN {X 0,Y 199.828,Z 412.693,A -85,B 0,C 180,E1 -21431.154,E2 -21431.154} C_VEL
LIN {X 0,Y 201.455,Z 403.382,A -85,B 0,C 180,E1 -21434.651,E2 -21434.651} C_VEL
LIN {X 0,Y 203.597,Z 392.434,A -85,B 0,C 180,E1 -21438.1,E2 -21438.1} C_VEL
LIN {X 0,Y 206.316,Z 379.294,A -85,B 0,C 180,E1 -21441.481,E2 -21441.481} C_VEL
LIN {X 0,Y 208.936,Z 366.503,A -85,B 0,C 180,E1 -21444.218,E2 -21444.218} C_VEL
LIN {X 0,Y 211.808,Z 351.502,A -85,B 0,C 180,E1 -21446.878,E2 -21446.878} C_VEL
LIN {X 0,Y 213.266,Z 344.202,A -85,B 0,C 180,E1 -21447.982,E2 -21447.982} C_VEL
LIN {X 0,Y 212.433,Z 339.067,A -85,B 0,C 180,E1 -21448.842,E2 -21448.842} C_VEL
LIN {X 0,Y 209.396,Z 325.775,A -85,B 0,C 180,E1 -21450.969,E2 -21450.969} C_VEL
LIN {X 0,Y 205.847,Z 313.839,A -85,B 0,C 180,E1 -21452.782,E2 -21452.782} C_VEL
LIN {X 0,Y 200.083,Z 297.237,A -85,B 0,C 180,E1 -21455.125,E2 -21455.125} C_VEL
LIN {X 0,Y 199.537,Z 295.257,A -85,B 0,C 180,E1 -21455.439,E2 -21455.439} C_VEL
LIN {X 0,Y 199.597,Z 295.252,A -85,B 0,C 180,E1 -21459.331,E2 -21459.331} C_VEL
LIN {X 0,Y 199.573,Z 295.253,A -85,B 0,C 180,E1 -21462.309,E2 -21462.309} C_VEL
LIN {X 0,Y 199.58,Z 295.252,A -85,B 0,C 180,E1 -21465.228,E2 -21465.228} C_VEL
LIN {X 0,Y 199.58,Z 295.247,A -85,B 0,C 180,E1 -21468.005,E2 -21468.005} C_VEL
LIN {X 0,Y 199.613,Z 295.246,A -85,B 0,C 180,E1 -21470.768,E2 -21470.768} C_VEL
LIN {X 0,Y 199.614,Z 295.244,A -85,B 0,C 180,E1 -21475.714,E2 -21475.714} C_VEL
LIN {X 0,Y 199.696,Z 295.234,A -85,B 0,C 180,E1 -21478.136,E2 -21478.136} C_VEL
LIN {X 0,Y 199.689,Z 295.236,A -85,B 0,C 180,E1 -21482.772,E2 -21482.772} C_VEL
LIN {X 0,Y 199.741,Z 295.225,A -85,B 0,C 180,E1 -21487.229,E2 -21487.229} C_VEL
LIN {X 0,Y 199.8,Z 295.221,A -85,B 0,C 180,E1 -21491.758,E2 -21491.758} C_VEL
LIN {X 0,Y 199.839,Z 295.213,A -85,B 0,C 180,E1 -21495.749,E2 -21495.749} C_VEL
LIN {X 0,Y 200.025,Z 295.194,A -85,B 0,C 180,E1 -21499.882,E2 -21499.882} C_VEL
LIN {X 0,Y 200.01,Z 295.193,A -85,B 0,C 180,E1 -21503.949,E2 -21503.949} C_VEL
LIN {X 0,Y 200.317,Z 295.159,A -85,B 0,C 180,E1 -21507.989,E2 -21507.989} C_VEL
LIN {X 0,Y 200.476,Z 295.136,A -85,B 0,C 180,E1 -21510,E2 -21510} C_VEL
LIN {X 0,Y 200.021,Z 295.195,A -85,B 0,C 180,E1 -21514.03,E2 -21514.03} C_VEL
LIN {X 0,Y 200.085,Z 295.184,A -85,B 0,C 180,E1 -21518.077,E2 -21518.077} C_VEL
LIN {X 0,Y 199.878,Z 295.211,A -85,B 0,C 180,E1 -21522.179,E2 -21522.179} C_VEL
LIN {X 0,Y 199.81,Z 295.217,A -85,B 0,C 180,E1 -21526.343,E2 -21526.343} C_VEL
LIN {X 0,Y 199.745,Z 295.227,A -85,B 0,C 180,E1 -21530.601,E2 -21530.601} C_VEL
LIN {X 0,Y 199.679,Z 295.235,A -85,B 0,C 180,E1 -21534.984,E2 -21534.984} C_VEL
LIN {X 0,Y 199.667,Z 295.239,A -85,B 0,C 180,E1 -21539.524,E2 -21539.524} C_VEL
LIN {X 0,Y 199.674,Z 295.235,A -85,B 0,C 180,E1 -21542.355,E2 -21542.355} C_VEL
LIN {X 0,Y 199.62,Z 295.243,A -85,B 0,C 180,E1 -21546.764,E2 -21546.764} C_VEL
LIN {X 0,Y 199.597,Z 295.247,A -85,B 0,C 180,E1 -21549.331,E2 -21549.331} C_VEL
LIN {X 0,Y 199.569,Z 295.246,A -85,B 0,C 180,E1 -21552.307,E2 -21552.307} C_VEL
LIN {X 0,Y 199.58,Z 295.25,A -85,B 0,C 180,E1 -21555.228,E2 -21555.228} C_VEL
LIN {X 0,Y 199.581,Z 295.247,A -85,B 0,C 180,E1 -21558.004,E2 -21558.004} C_VEL
LIN {X 0,Y 199.613,Z 295.243,A -85,B 0,C 180,E1 -21560.767,E2 -21560.767} C_VEL
LIN {X 0,Y 199.615,Z 295.243,A -85,B 0,C 180,E1 -21565.713,E2 -21565.713} C_VEL
LIN {X 0,Y 199.696,Z 295.232,A -85,B 0,C 180,E1 -21568.136,E2 -21568.136} C_VEL
LIN {X 0,Y 199.689,Z 295.237,A -85,B 0,C 180,E1 -21572.771,E2 -21572.771} C_VEL
LIN {X 0,Y 199.741,Z 295.224,A -85,B 0,C 180,E1 -21577.229,E2 -21577.229} C_VEL
LIN {X 0,Y 199.8,Z 295.221,A -85,B 0,C 180,E1 -21581.757,E2 -21581.757} C_VEL
LIN {X 0,Y 199.839,Z 295.212,A -85,B 0,C 180,E1 -21585.748,E2 -21585.748} C_VEL
LIN {X 0,Y 200.025,Z 295.194,A -85,B 0,C 180,E1 -21589.881,E2 -21589.881} C_VEL
LIN {X 0,Y 200.013,Z 295.193,A -85,B 0,C 180,E1 -21593.949,E2 -21593.949} C_VEL
LIN {X 0,Y 200.32,Z 295.159,A -85,B 0,C 180,E1 -21597.989,E2 -21597.989} C_VEL
LIN {X 0,Y 200.474,Z 295.138,A -85,B 0,C 180,E1 -21600,E2 -21600} C_VEL
LIN {X 0,Y 200.024,Z 295.195,A -85,B 0,C 180,E1 -21604.029,E2 -21604.029} C_VEL
LIN {X 0,Y 200.08,Z 295.186,A -85,B 0,C 180,E1 -21608.077,E2 -21608.077} C_VEL
LIN {X 0,Y 199.882,Z 295.211,A -85,B 0,C 180,E1 -21612.178,E2 -21612.178} C_VEL
LIN {X 0,Y 199.808,Z 295.218,A -85,B 0,C 180,E1 -21616.343,E2 -21616.343} C_VEL
LIN {X 0,Y 199.695,Z 295.234,A -85,B 0,C 180,E1 -21620.605,E2 -21620.605} C_VEL
LIN {X 0,Y 199.795,Z 295.328,A -85,B 0,C 180,E1 -21624.62,E2 -21624.62} C_VEL
LIN {X 0,Y 200.232,Z 299.009,A -85,B 0,C 180,E1 -21629.431,E2 -21629.431} C_VEL
LIN {X 0,Y 200.846,Z 302.72,A -85,B 0,C 180,E1 -21634.046,E2 -21634.046} C_VEL
LIN {X 0,Y 201.67,Z 306.797,A -85,B 0,C 180,E1 -21638.849,E2 -21638.849} C_VEL
LIN {X 0,Y 202.589,Z 310.71,A -85,B 0,C 180,E1 -21643.238,E2 -21643.238} C_VEL
LIN {X 0,Y 202.894,Z 313.296,A -85,B 0,C 180,E1 -21646.011,E2 -21646.011} C_VEL
LIN {X 0,Y 205.618,Z 325.965,A -85,B 0,C 180,E1 -21647.476,E2 -21647.476} C_VEL
LIN {X 0,Y 208.396,Z 342.395,A -85,B 0,C 180,E1 -21649.583,E2 -21649.583} C_VEL
LIN {X 0,Y 210.851,Z 358.387,A -85,B 0,C 180,E1 -21651.948,E2 -21651.948} C_VEL
LIN {X 0,Y 212.88,Z 372.904,A -85,B 0,C 180,E1 -21654.394,E2 -21654.394} C_VEL
LIN {X 0,Y 214.639,Z 386.606,A -85,B 0,C 180,E1 -21657.019,E2 -21657.019} C_VEL
LIN {X 0,Y 211.001,Z 400.209,A -85,B 0,C 180,E1 -21659.749,E2 -21659.749} C_VEL
LIN {X 0,Y 207.523,Z 412.586,A -85,B 0,C 180,E1 -21662.794,E2 -21662.794} C_VEL
LIN {X 0,Y 204.419,Z 423.803,A -85,B 0,C 180,E1 -21666.173,E2 -21666.173} C_VEL
LIN {X 0,Y 201.953,Z 433.233,A -85,B 0,C 180,E1 -21669.635,E2 -21669.635} C_VEL
LIN {X 0,Y 200.153,Z 441.16,A -85,B 0,C 180,E1 -21673.161,E2 -21673.161} C_VEL
LIN {X 0,Y 198.922,Z 447.74,A -85,B 0,C 180,E1 -21676.723,E2 -21676.723} C_VEL
LIN {X 0,Y 198.665,Z 449.551,A -85,B 0,C 180,E1 -21677.821,E2 -21677.821} C_VEL
LIN {X 0,Y 197.697,Z 451.792,A -85,B 0,C 180,E1 -21679.384,E2 -21679.384} C_VEL
LIN {X 0,Y 194.568,Z 454.76,A -85,B 0,C 180,E1 -21681.992,E2 -21681.992} C_VEL
LIN {X 0,Y 192.048,Z 456.772,A -85,B 0,C 180,E1 -21684.165,E2 -21684.165} C_VEL
LIN {X 0,Y 190.953,Z 458.207,A -85,B 0,C 180,E1 -21685.87,E2 -21685.87} C_VEL
LIN {X 0,Y 190.847,Z 458.666,A -85,B 0,C 180,E1 -21686.449,E2 -21686.449} C_VEL
LIN {X 0,Y 190.871,Z 461.264,A -85,B 0,C 180,E1 -21690,E2 -21690} C_VEL
LIN {X 0,Y 190.596,Z 463.089,A -85,B 0,C 180,E1 -21694.229,E2 -21694.229} C_VEL
LIN {X 0,Y 190.541,Z 463.827,A -85,B 0,C 180,E1 -21698.484,E2 -21698.484} C_VEL
LIN {X 0,Y 191.171,Z 463.636,A -85,B 0,C 180,E1 -21702.743,E2 -21702.743} C_VEL
LIN {X 0,Y 193.989,Z 461.702,A -85,B 0,C 180,E1 -21709.03,E2 -21709.03} C_VEL
LIN {X 0,Y 199.184,Z 457.958,A -85,B 0,C 180,E1 -21715.05,E2 -21715.05} C_VEL
LIN {X 0,Y 206.693,Z 452.607,A -85,B 0,C 180,E1 -21720.666,E2 -21720.666} C_VEL
LIN {X 0,Y 214.894,Z 446.991,A -85,B 0,C 180,E1 -21724.913,E2 -21724.913} C_VEL
LIN {X 0,Y 224.602,Z 440.313,A -85,B 0,C 180,E1 -21728.743,E2 -21728.743} C_VEL
LIN {X 0,Y 235.718,Z 432.587,A -85,B 0,C 180,E1 -21732.133,E2 -21732.133} C_VEL
LIN {X 0,Y 246.387,Z 425.103,A -85,B 0,C 180,E1 -21734.698,E2 -21734.698} C_VEL
LIN {X 0,Y 245.854,Z 425.359,A -85,B 0,C 180,E1 -21735.129,E2 -21735.129} C_VEL
LIN {X 0,Y 235.604,Z 431.217,A -85,B 0,C 180,E1 -21737.843,E2 -21737.843} C_VEL
LIN {X 0,Y 225.073,Z 436.837,A -85,B 0,C 180,E1 -21741.354,E2 -21741.354} C_VEL
LIN {X 0,Y 217.589,Z 440.461,A -85,B 0,C 180,E1 -21744.452,E2 -21744.452} C_VEL
LIN {X 0,Y 211.02,Z 443.329,A -85,B 0,C 180,E1 -21747.8,E2 -21747.8} C_VEL
LIN {X 0,Y 202.837,Z 446.022,A -85,B 0,C 180,E1 -21753.229,E2 -21753.229} C_VEL
LIN {X 0,Y 198.573,Z 446.799,A -85,B 0,C 180,E1 -21757.088,E2 -21757.088} C_VEL
LIN {X 0,Y 195.285,Z 446.588,A -85,B 0,C 180,E1 -21761.102,E2 -21761.102} C_VEL
LIN {X 0,Y 192.909,Z 445.427,A -85,B 0,C 180,E1 -21765.226,E2 -21765.226} C_VEL
LIN {X 0,Y 191.487,Z 443.275,A -85,B 0,C 180,E1 -21769.426,E2 -21769.426} C_VEL
LIN {X 0,Y 190.773,Z 440.046,A -85,B 0,C 180,E1 -21773.655,E2 -21773.655} C_VEL
LIN {X 0,Y 190.592,Z 435.641,A -85,B 0,C 180,E1 -21777.887,E2 -21777.887} C_VEL
LIN {X 0,Y 190.79,Z 429.988,A -85,B 0,C 180,E1 -21782.112,E2 -21782.112} C_VEL
LIN {X 0,Y 191.46,Z 422.919,A -85,B 0,C 180,E1 -21786.323,E2 -21786.323} C_VEL
LIN {X 0,Y 192.564,Z 413.907,A -85,B 0,C 180,E1 -21790.679,E2 -21790.679} C_VEL
LIN {X 0,Y 194.303,Z 403.744,A -85,B 0,C 180,E1 -21794.667,E2 -21794.667} C_VEL
LIN {X 0,Y 196.501,Z 392.758,A -85,B 0,C 180,E1 -21798.238,E2 -21798.238} C_VEL
LIN {X 0,Y 199.243,Z 379.708,A -85,B 0,C 180,E1 -21801.739,E2 -21801.739} C_VEL
LIN {X 0,Y 201.844,Z 367.71,A -85,B 0,C 180,E1 -21804.424,E2 -21804.424} C_VEL
LIN {X 0,Y 204.344,Z 354.884,A -85,B 0,C 180,E1 -21806.835,E2 -21806.835} C_VEL
LIN {X 0,Y 206.349,Z 344.573,A -85,B 0,C 180,E1 -21808.479,E2 -21808.479} C_VEL
LIN {X 0,Y 203.512,Z 331.149,A -85,B 0,C 180,E1 -21810.792,E2 -21810.792} C_VEL
LIN {X 0,Y 200.972,Z 321.489,A -85,B 0,C 180,E1 -21812.367,E2 -21812.367} C_VEL
LIN {X 0,Y 195.813,Z 305.757,A -85,B 0,C 180,E1 -21814.761,E2 -21814.761} C_VEL
LIN {X 0,Y 192.5,Z 296.133,A -85,B 0,C 180,E1 -21816.144,E2 -21816.144} C_VEL
LIN {X 0,Y 192.51,Z 296.135,A -85,B 0,C 180,E1 -21821.082,E2 -21821.082} C_VEL
LIN {X 0,Y 192.492,Z 296.133,A -85,B 0,C 180,E1 -21826.076,E2 -21826.076} C_VEL
LIN {X 0,Y 192.52,Z 296.128,A -85,B 0,C 180,E1 -21830.051,E2 -21830.051} C_VEL
LIN {X 0,Y 192.563,Z 296.123,A -85,B 0,C 180,E1 -21834.271,E2 -21834.271} C_VEL
LIN {X 0,Y 192.61,Z 296.118,A -85,B 0,C 180,E1 -21837.06,E2 -21837.06} C_VEL
LIN {X 0,Y 192.663,Z 296.109,A -85,B 0,C 180,E1 -21841.692,E2 -21841.692} C_VEL
LIN {X 0,Y 192.709,Z 296.103,A -85,B 0,C 180,E1 -21846.349,E2 -21846.349} C_VEL
LIN {X 0,Y 192.735,Z 296.1,A -85,B 0,C 180,E1 -21851.458,E2 -21851.458} C_VEL
LIN {X 0,Y 192.767,Z 296.093,A -85,B 0,C 180,E1 -21855.214,E2 -21855.214} C_VEL
LIN {X 0,Y 192.948,Z 296.075,A -85,B 0,C 180,E1 -21859.567,E2 -21859.567} C_VEL
LIN {X 0,Y 192.974,Z 296.068,A -85,B 0,C 180,E1 -21863.727,E2 -21863.727} C_VEL
LIN {X 0,Y 193.258,Z 296.038,A -85,B 0,C 180,E1 -21867.916,E2 -21867.916} C_VEL
LIN {X 0,Y 193.44,Z 296.012,A -85,B 0,C 180,E1 -21870,E2 -21870} C_VEL
LIN {X 0,Y 192.967,Z 296.073,A -85,B 0,C 180,E1 -21874.177,E2 -21874.177} C_VEL
LIN {X 0,Y 193.034,Z 296.061,A -85,B 0,C 180,E1 -21878.374,E2 -21878.374} C_VEL
LIN {X 0,Y 192.806,Z 296.092,A -85,B 0,C 180,E1 -21882.633,E2 -21882.633} C_VEL
LIN {X 0,Y 192.775,Z 296.094,A -85,B 0,C 180,E1 -21886.957,E2 -21886.957} C_VEL
LIN {X 0,Y 192.671,Z 296.111,A -85,B 0,C 180,E1 -21891.393,E2 -21891.393} C_VEL
LIN {X 0,Y 192.672,Z 296.107,A -85,B 0,C 180,E1 -21894.227,E2 -21894.227} C_VEL
LIN {X 0,Y 192.647,Z 296.112,A -85,B 0,C 180,E1 -21898.889,E2 -21898.889} C_VEL
LIN {X 0,Y 192.599,Z 296.117,A -85,B 0,C 180,E1 -21903.186,E2 -21903.186} C_VEL
LIN {X 0,Y 192.544,Z 296.125,A -85,B 0,C 180,E1 -21908.354,E2 -21908.354} C_VEL
LIN {X 0,Y 192.488,Z 296.13,A -85,B 0,C 180,E1 -21913.094,E2 -21913.094} C_VEL
LIN {X 0,Y 192.492,Z 296.134,A -85,B 0,C 180,E1 -21916.905,E2 -21916.905} C_VEL
LIN {X 0,Y 192.554,Z 296.121,A -85,B 0,C 180,E1 -21921.648,E2 -21921.648} C_VEL
LIN {X 0,Y 192.6,Z 296.118,A -85,B 0,C 180,E1 -21926.814,E2 -21926.814} C_VEL
LIN {X 0,Y 192.664,Z 296.109,A -85,B 0,C 180,E1 -21931.691,E2 -21931.691} C_VEL
LIN {X 0,Y 192.709,Z 296.104,A -85,B 0,C 180,E1 -21936.348,E2 -21936.348} C_VEL
LIN {X 0,Y 192.735,Z 296.101,A -85,B 0,C 180,E1 -21941.457,E2 -21941.457} C_VEL
LIN {X 0,Y 192.768,Z 296.092,A -85,B 0,C 180,E1 -21945.213,E2 -21945.213} C_VEL
LIN {X 0,Y 192.948,Z 296.074,A -85,B 0,C 180,E1 -21949.566,E2 -21949.566} C_VEL
LIN {X 0,Y 192.976,Z 296.068,A -85,B 0,C 180,E1 -21953.727,E2 -21953.727} C_VEL
LIN {X 0,Y 193.261,Z 296.038,A -85,B 0,C 180,E1 -21957.915,E2 -21957.915} C_VEL
LIN {X 0,Y 193.438,Z 296.014,A -85,B 0,C 180,E1 -21959.999,E2 -21959.999} C_VEL
LIN {X 0,Y 192.969,Z 296.073,A -85,B 0,C 180,E1 -21964.177,E2 -21964.177} C_VEL
LIN {X 0,Y 193.03,Z 296.063,A -85,B 0,C 180,E1 -21968.374,E2 -21968.374} C_VEL
LIN {X 0,Y 192.808,Z 296.091,A -85,B 0,C 180,E1 -21972.632,E2 -21972.632} C_VEL
LIN {X 0,Y 192.76,Z 296.096,A -85,B 0,C 180,E1 -21976.958,E2 -21976.958} C_VEL
LIN {X 0,Y 192.628,Z 296.117,A -85,B 0,C 180,E1 -21981.398,E2 -21981.398} C_VEL
LIN {X 0,Y 192.754,Z 296.258,A -85,B 0,C 180,E1 -21984.5,E2 -21984.5} C_VEL
LIN {X 0,Y 193.17,Z 299.728,A -85,B 0,C 180,E1 -21989.169,E2 -21989.169} C_VEL
LIN {X 0,Y 193.701,Z 303.047,A -85,B 0,C 180,E1 -21993.435,E2 -21993.435} C_VEL
LIN {X 0,Y 194.409,Z 306.703,A -85,B 0,C 180,E1 -21997.919,E2 -21997.919} C_VEL
LIN {X 0,Y 195.002,Z 309.162,A -85,B 0,C 180,E1 -22000.812,E2 -22000.812} C_VEL
LIN {X 0,Y 195.804,Z 312.899,A -85,B 0,C 180,E1 -22005.058,E2 -22005.058} C_VEL
LIN {X 0,Y 198.551,Z 324.766,A -85,B 0,C 180,E1 -22006.519,E2 -22006.519} C_VEL
LIN {X 0,Y 201.243,Z 340.982,A -85,B 0,C 180,E1 -22008.661,E2 -22008.661} C_VEL
LIN {X 0,Y 203.622,Z 356.951,A -85,B 0,C 180,E1 -22011.085,E2 -22011.085} C_VEL
LIN {X 0,Y 205.673,Z 371.716,A -85,B 0,C 180,E1 -22013.652,E2 -22013.652} C_VEL
LIN {X 0,Y 207.338,Z 385.127,A -85,B 0,C 180,E1 -22016.285,E2 -22016.285} C_VEL
LIN {X 0,Y 207.395,Z 388.013,A -85,B 0,C 180,E1 -22016.877,E2 -22016.877} C_VEL
LIN {X 0,Y 203.819,Z 400.598,A -85,B 0,C 180,E1 -22019.545,E2 -22019.545} C_VEL
LIN {X 0,Y 200.683,Z 411.562,A -85,B 0,C 180,E1 -22022.353,E2 -22022.353} C_VEL
LIN {X 0,Y 197.491,Z 422.819,A -85,B 0,C 180,E1 -22025.842,E2 -22025.842} C_VEL
LIN {X 0,Y 194.819,Z 432.971,A -85,B 0,C 180,E1 -22029.707,E2 -22029.707} C_VEL
LIN {X 0,Y 192.889,Z 441.289,A -85,B 0,C 180,E1 -22033.598,E2 -22033.598} C_VEL
LIN {X 0,Y 191.634,Z 448.523,A -85,B 0,C 180,E1 -22037.814,E2 -22037.814} C_VEL
LIN {X 0,Y 191.105,Z 453.641,A -85,B 0,C 180,E1 -22041.541,E2 -22041.541} C_VEL
LIN {X 0,Y 190.973,Z 456.933,A -85,B 0,C 180,E1 -22044.498,E2 -22044.498} C_VEL
LIN {X 0,Y 190.847,Z 458.666,A -85,B 0,C 180,E1 -22046.449,E2 -22046.449} C_VEL
LIN {X 0,Y 190.488,Z 459.585,A -85,B 0,C 180,E1 -22047.598,E2 -22047.598} C_VEL
LIN {X 0,Y 188.495,Z 460.82,A -85,B 0,C 180,E1 -22049.881,E2 -22049.881} C_VEL
LIN {X 0,Y 184.703,Z 461.952,A -85,B 0,C 180,E1 -22053.373,E2 -22053.373} C_VEL
LIN {X 0,Y 183.596,Z 462.384,A -85,B 0,C 180,E1 -22055.208,E2 -22055.208} C_VEL
LIN {X 0,Y 183.482,Z 462.535,A -85,B 0,C 180,E1 -22055.83,E2 -22055.83} C_VEL
LIN {X 0,Y 183.779,Z 463.17,A -85,B 0,C 180,E1 -22061.023,E2 -22061.023} C_VEL
LIN {X 0,Y 184.975,Z 462.747,A -85,B 0,C 180,E1 -22065.424,E2 -22065.424} C_VEL
LIN {X 0,Y 187.807,Z 461.109,A -85,B 0,C 180,E1 -22070.687,E2 -22070.687} C_VEL
LIN {X 0,Y 192.749,Z 458.155,A -85,B 0,C 180,E1 -22075.947,E2 -22075.947} C_VEL
LIN {X 0,Y 200.644,Z 453.291,A -85,B 0,C 180,E1 -22081.696,E2 -22081.696} C_VEL
LIN {X 0,Y 209.197,Z 448.089,A -85,B 0,C 180,E1 -22086.009,E2 -22086.009} C_VEL
LIN {X 0,Y 219.246,Z 441.94,A -85,B 0,C 180,E1 -22089.875,E2 -22089.875} C_VEL
LIN {X 0,Y 230.728,Z 434.807,A -85,B 0,C 180,E1 -22093.264,E2 -22093.264} C_VEL
LIN {X 0,Y 237.04,Z 430.804,A -85,B 0,C 180,E1 -22094.798,E2 -22094.798} C_VEL
LIN {X 0,Y 236.408,Z 431.05,A -85,B 0,C 180,E1 -22095.226,E2 -22095.226} C_VEL
LIN {X 0,Y 223.321,Z 437.43,A -85,B 0,C 180,E1 -22099.051,E2 -22099.051} C_VEL
LIN {X 0,Y 215.833,Z 440.765,A -85,B 0,C 180,E1 -22101.781,E2 -22101.781} C_VEL
LIN {X 0,Y 208.506,Z 443.622,A -85,B 0,C 180,E1 -22105.04,E2 -22105.04} C_VEL
LIN {X 0,Y 199.223,Z 446.54,A -85,B 0,C 180,E1 -22110.405,E2 -22110.405} C_VEL
LIN {X 0,Y 192.373,Z 447.541,A -85,B 0,C 180,E1 -22115.971,E2 -22115.971} C_VEL
LIN {X 0,Y 188.564,Z 447.147,A -85,B 0,C 180,E1 -22120.401,E2 -22120.401} C_VEL
LIN {X 0,Y 185.999,Z 445.747,A -85,B 0,C 180,E1 -22124.663,E2 -22124.663} C_VEL
LIN {X 0,Y 184.472,Z 443.36,A -85,B 0,C 180,E1 -22129.019,E2 -22129.019} C_VEL
LIN {X 0,Y 183.701,Z 439.938,A -85,B 0,C 180,E1 -22133.41,E2 -22133.41} C_VEL
LIN {X 0,Y 183.51,Z 435.383,A -85,B 0,C 180,E1 -22137.806,E2 -22137.806} C_VEL
LIN {X 0,Y 183.731,Z 429.534,A -85,B 0,C 180,E1 -22142.193,E2 -22142.193} C_VEL
LIN {X 0,Y 184.208,Z 424.211,A -85,B 0,C 180,E1 -22145.474,E2 -22145.474} C_VEL
LIN {X 0,Y 185.186,Z 415.708,A -85,B 0,C 180,E1 -22149.834,E2 -22149.834} C_VEL
LIN {X 0,Y 186.876,Z 405.447,A -85,B 0,C 180,E1 -22154.15,E2 -22154.15} C_VEL
LIN {X 0,Y 189.037,Z 394.732,A -85,B 0,C 180,E1 -22157.862,E2 -22157.862} C_VEL
LIN {X 0,Y 191.732,Z 382.019,A -85,B 0,C 180,E1 -22161.504,E2 -22161.504} C_VEL
LIN {X 0,Y 194.824,Z 367.972,A -85,B 0,C 180,E1 -22164.794,E2 -22164.794} C_VEL
LIN {X 0,Y 197.683,Z 353.864,A -85,B 0,C 180,E1 -22167.528,E2 -22167.528} C_VEL
LIN {X 0,Y 199.342,Z 345.032,A -85,B 0,C 180,E1 -22168.998,E2 -22168.998} C_VEL
LIN {X 0,Y 196.489,Z 331.836,A -85,B 0,C 180,E1 -22171.355,E2 -22171.355} C_VEL
LIN {X 0,Y 193.68,Z 321.539,A -85,B 0,C 180,E1 -22173.097,E2 -22173.097} C_VEL
LIN {X 0,Y 188.79,Z 306.611,A -85,B 0,C 180,E1 -22175.478,E2 -22175.478} C_VEL
LIN {X 0,Y 185.462,Z 297.014,A -85,B 0,C 180,E1 -22176.907,E2 -22176.907} C_VEL
LIN {X 0,Y 185.466,Z 297.013,A -85,B 0,C 180,E1 -22180.722,E2 -22180.722} C_VEL
LIN {X 0,Y 185.461,Z 297.009,A -85,B 0,C 180,E1 -22186.055,E2 -22186.055} C_VEL
LIN {X 0,Y 185.47,Z 297.006,A -85,B 0,C 180,E1 -22189.896,E2 -22189.896} C_VEL
LIN {X 0,Y 185.509,Z 297.003,A -85,B 0,C 180,E1 -22192.711,E2 -22192.711} C_VEL
LIN {X 0,Y 185.545,Z 296.997,A -85,B 0,C 180,E1 -22197.975,E2 -22197.975} C_VEL
LIN {X 0,Y 185.583,Z 296.993,A -85,B 0,C 180,E1 -22200.577,E2 -22200.577} C_VEL
LIN {X 0,Y 185.59,Z 296.988,A -85,B 0,C 180,E1 -22205.383,E2 -22205.383} C_VEL
LIN {X 0,Y 185.678,Z 296.98,A -85,B 0,C 180,E1 -22211.133,E2 -22211.133} C_VEL
LIN {X 0,Y 185.699,Z 296.975,A -85,B 0,C 180,E1 -22214.638,E2 -22214.638} C_VEL
LIN {X 0,Y 185.891,Z 296.953,A -85,B 0,C 180,E1 -22219.419,E2 -22219.419} C_VEL
LIN {X 0,Y 185.938,Z 296.943,A -85,B 0,C 180,E1 -22223.489,E2 -22223.489} C_VEL
LIN {X 0,Y 186.202,Z 296.917,A -85,B 0,C 180,E1 -22227.837,E2 -22227.837} C_VEL
LIN {X 0,Y 186.404,Z 296.888,A -85,B 0,C 180,E1 -22230,E2 -22230} C_VEL
LIN {X 0,Y 185.914,Z 296.951,A -85,B 0,C 180,E1 -22234.336,E2 -22234.336} C_VEL
LIN {X 0,Y 185.982,Z 296.939,A -85,B 0,C 180,E1 -22238.694,E2 -22238.694} C_VEL
LIN {X 0,Y 185.733,Z 296.973,A -85,B 0,C 180,E1 -22243.123,E2 -22243.123} C_VEL
LIN {X 0,Y 185.721,Z 296.973,A -85,B 0,C 180,E1 -22247.622,E2 -22247.622} C_VEL
LIN {X 0,Y 185.62,Z 296.987,A -85,B 0,C 180,E1 -22252.249,E2 -22252.249} C_VEL
LIN {X 0,Y 185.564,Z 296.991,A -85,B 0,C 180,E1 -22257.032,E2 -22257.032} C_VEL
LIN {X 0,Y 185.58,Z 296.994,A -85,B 0,C 180,E1 -22259.493,E2 -22259.493} C_VEL
LIN {X 0,Y 185.5,Z 296.998,A -85,B 0,C 180,E1 -22264.632,E2 -22264.632} C_VEL
LIN {X 0,Y 185.502,Z 297.004,A -85,B 0,C 180,E1 -22267.314,E2 -22267.314} C_VEL
LIN {X 0,Y 185.464,Z 297.007,A -85,B 0,C 180,E1 -22270.721,E2 -22270.721} C_VEL
LIN {X 0,Y 185.461,Z 297.007,A -85,B 0,C 180,E1 -22276.055,E2 -22276.055} C_VEL
LIN {X 0,Y 185.47,Z 297.003,A -85,B 0,C 180,E1 -22279.895,E2 -22279.895} C_VEL
LIN {X 0,Y 185.509,Z 297.001,A -85,B 0,C 180,E1 -22282.711,E2 -22282.711} C_VEL
LIN {X 0,Y 185.545,Z 296.994,A -85,B 0,C 180,E1 -22287.974,E2 -22287.974} C_VEL
LIN {X 0,Y 185.583,Z 296.991,A -85,B 0,C 180,E1 -22290.576,E2 -22290.576} C_VEL
LIN {X 0,Y 185.591,Z 296.989,A -85,B 0,C 180,E1 -22295.382,E2 -22295.382} C_VEL
LIN {X 0,Y 185.678,Z 296.98,A -85,B 0,C 180,E1 -22301.133,E2 -22301.133} C_VEL
LIN {X 0,Y 185.699,Z 296.974,A -85,B 0,C 180,E1 -22304.637,E2 -22304.637} C_VEL
LIN {X 0,Y 185.891,Z 296.953,A -85,B 0,C 180,E1 -22309.418,E2 -22309.418} C_VEL
LIN {X 0,Y 185.94,Z 296.944,A -85,B 0,C 180,E1 -22313.489,E2 -22313.489} C_VEL
LIN {X 0,Y 186.205,Z 296.916,A -85,B 0,C 180,E1 -22317.836,E2 -22317.836} C_VEL
LIN {X 0,Y 186.403,Z 296.89,A -85,B 0,C 180,E1 -22319.999,E2 -22319.999} C_VEL
LIN {X 0,Y 185.916,Z 296.951,A -85,B 0,C 180,E1 -22324.335,E2 -22324.335} C_VEL
LIN {X 0,Y 185.979,Z 296.94,A -85,B 0,C 180,E1 -22328.693,E2 -22328.693} C_VEL
LIN {X 0,Y 185.734,Z 296.973,A -85,B 0,C 180,E1 -22333.122,E2 -22333.122} C_VEL
LIN {X 0,Y 185.693,Z 296.977,A -85,B 0,C 180,E1 -22337.624,E2 -22337.624} C_VEL
LIN {X 0,Y 185.718,Z 297.111,A -85,B 0,C 180,E1 -22344.301,E2 -22344.301} C_VEL
LIN {X 0,Y 186.174,Z 301.037,A -85,B 0,C 180,E1 -22349.744,E2 -22349.744} C_VEL
LIN {X 0,Y 186.984,Z 305.554,A -85,B 0,C 180,E1 -22355.632,E2 -22355.632} C_VEL
LIN {X 0,Y 187.678,Z 308.709,A -85,B 0,C 180,E1 -22359.538,E2 -22359.538} C_VEL
LIN {X 0,Y 188.585,Z 312.492,A -85,B 0,C 180,E1 -22364.048,E2 -22364.048} C_VEL
LIN {X 0,Y 192.04,Z 326.732,A -85,B 0,C 180,E1 -22365.946,E2 -22365.946} C_VEL
LIN {X 0,Y 194.735,Z 343.988,A -85,B 0,C 180,E1 -22368.368,E2 -22368.368} C_VEL
LIN {X 0,Y 196.985,Z 359.559,A -85,B 0,C 180,E1 -22370.894,E2 -22370.894} C_VEL
LIN {X 0,Y 198.904,Z 374.029,A -85,B 0,C 180,E1 -22373.565,E2 -22373.565} C_VEL
LIN {X 0,Y 200.397,Z 386.571,A -85,B 0,C 180,E1 -22376.169,E2 -22376.169} C_VEL
LIN {X 0,Y 200.43,Z 388.019,A -85,B 0,C 180,E1 -22376.477,E2 -22376.477} C_VEL
LIN {X 0,Y 196.452,Z 401.544,A -85,B 0,C 180,E1 -22379.493,E2 -22379.493} C_VEL
LIN {X 0,Y 192.802,Z 413.864,A -85,B 0,C 180,E1 -22382.893,E2 -22382.893} C_VEL
LIN {X 0,Y 189.811,Z 424.658,A -85,B 0,C 180,E1 -22386.544,E2 -22386.544} C_VEL
LIN {X 0,Y 187.407,Z 433.71,A -85,B 0,C 180,E1 -22390.274,E2 -22390.274} C_VEL
LIN {X 0,Y 185.504,Z 442.296,A -85,B 0,C 180,E1 -22394.621,E2 -22394.621} C_VEL
LIN {X 0,Y 184.408,Z 449.212,A -85,B 0,C 180,E1 -22399.015,E2 -22399.015} C_VEL
LIN {X 0,Y 184.007,Z 454.65,A -85,B 0,C 180,E1 -22403.42,E2 -22403.42} C_VEL
LIN {X 0,Y 183.842,Z 457.544,A -85,B 0,C 180,E1 -22406.505,E2 -22406.505} C_VEL
LIN {X 0,Y 183.865,Z 460.109,A -85,B 0,C 180,E1 -22410,E2 -22410} C_VEL
LIN {X 0,Y 183.571,Z 462.124,A -85,B 0,C 180,E1 -22414.391,E2 -22414.391} C_VEL
LIN {X 0,Y 183.482,Z 462.535,A -85,B 0,C 180,E1 -22415.83,E2 -22415.83} C_VEL
LIN {X 0,Y 182.773,Z 462.842,A -85,B 0,C 180,E1 -22417.662,E2 -22417.662} C_VEL
LIN {X 0,Y 180.129,Z 462.83,A -85,B 0,C 180,E1 -22420.681,E2 -22420.681} C_VEL
LIN {X 0,Y 178.211,Z 462.566,A -85,B 0,C 180,E1 -22423.154,E2 -22423.154} C_VEL
LIN {X 0,Y 177.785,Z 462.329,A -85,B 0,C 180,E1 -22425.057,E2 -22425.057} C_VEL
LIN {X 0,Y 177.955,Z 462.249,A -85,B 0,C 180,E1 -22425.691,E2 -22425.691} C_VEL
LIN {X 0,Y 180.888,Z 460.972,A -85,B 0,C 180,E1 -22431.179,E2 -22431.179} C_VEL
LIN {X 0,Y 186.358,Z 458.295,A -85,B 0,C 180,E1 -22436.907,E2 -22436.907} C_VEL
LIN {X 0,Y 194.652,Z 453.891,A -85,B 0,C 180,E1 -22442.792,E2 -22442.792} C_VEL
LIN {X 0,Y 203.563,Z 449.157,A -85,B 0,C 180,E1 -22447.17,E2 -22447.17} C_VEL
LIN {X 0,Y 213.972,Z 443.466,A -85,B 0,C 180,E1 -22451.065,E2 -22451.065} C_VEL
LIN {X 0,Y 226.992,Z 436.212,A -85,B 0,C 180,E1 -22454.75,E2 -22454.75} C_VEL
LIN {X 0,Y 225.871,Z 436.572,A -85,B 0,C 180,E1 -22455.646,E2 -22455.646} C_VEL
LIN {X 0,Y 214.686,Z 441.14,A -85,B 0,C 180,E1 -22459.102,E2 -22459.102} C_VEL
LIN {X 0,Y 206.565,Z 444.044,A -85,B 0,C 180,E1 -22462.236,E2 -22462.236} C_VEL
LIN {X 0,Y 199.397,Z 446.241,A -85,B 0,C 180,E1 -22465.672,E2 -22465.672} C_VEL
LIN {X 0,Y 190.339,Z 448.074,A -85,B 0,C 180,E1 -22471.315,E2 -22471.315} C_VEL
LIN {X 0,Y 185.583,Z 448.291,A -85,B 0,C 180,E1 -22475.382,E2 -22475.382} C_VEL
LIN {X 0,Y 181.859,Z 447.596,A -85,B 0,C 180,E1 -22479.647,E2 -22479.647} C_VEL
LIN {X 0,Y 179.11,Z 446.013,A -85,B 0,C 180,E1 -22484.058,E2 -22484.058} C_VEL
LIN {X 0,Y 177.481,Z 443.41,A -85,B 0,C 180,E1 -22488.581,E2 -22488.581} C_VEL
LIN {X 0,Y 176.639,Z 439.761,A -85,B 0,C 180,E1 -22493.145,E2 -22493.145} C_VEL
LIN {X 0,Y 176.431,Z 434.997,A -85,B 0,C 180,E1 -22497.718,E2 -22497.718} C_VEL
LIN {X 0,Y 176.566,Z 430.594,A -85,B 0,C 180,E1 -22501.141,E2 -22501.141} C_VEL
LIN {X 0,Y 177.157,Z 423.483,A -85,B 0,C 180,E1 -22505.692,E2 -22505.692} C_VEL
LIN {X 0,Y 178.2,Z 414.793,A -85,B 0,C 180,E1 -22510.223,E2 -22510.223} C_VEL
LIN {X 0,Y 179.996,Z 404.245,A -85,B 0,C 180,E1 -22514.703,E2 -22514.703} C_VEL
LIN {X 0,Y 182.275,Z 393.265,A -85,B 0,C 180,E1 -22518.548,E2 -22518.548} C_VEL
LIN {X 0,Y 184.885,Z 381.277,A -85,B 0,C 180,E1 -22522.048,E2 -22522.048} C_VEL
LIN {X 0,Y 187.829,Z 368.204,A -85,B 0,C 180,E1 -22525.19,E2 -22525.19} C_VEL
LIN {X 0,Y 190.875,Z 353.541,A -85,B 0,C 180,E1 -22528.11,E2 -22528.11} C_VEL
LIN {X 0,Y 192.288,Z 346.792,A -85,B 0,C 180,E1 -22529.266,E2 -22529.266} C_VEL
LIN {X 0,Y 190.981,Z 339.043,A -85,B 0,C 180,E1 -22530.728,E2 -22530.728} C_VEL
LIN {X 0,Y 188.177,Z 327.482,A -85,B 0,C 180,E1 -22532.825,E2 -22532.825} C_VEL
LIN {X 0,Y 182.937,Z 310.909,A -85,B 0,C 180,E1 -22535.68,E2 -22535.68} C_VEL
LIN {X 0,Y 178.379,Z 297.895,A -85,B 0,C 180,E1 -22537.775,E2 -22537.775} C_VEL
LIN {X 0,Y 178.398,Z 297.891,A -85,B 0,C 180,E1 -22542.046,E2 -22542.046} C_VEL
LIN {X 0,Y 178.395,Z 297.891,A -85,B 0,C 180,E1 -22545.164,E2 -22545.164} C_VEL
LIN {X 0,Y 178.405,Z 297.886,A -85,B 0,C 180,E1 -22548.459,E2 -22548.459} C_VEL
LIN {X 0,Y 178.425,Z 297.883,A -85,B 0,C 180,E1 -22553.783,E2 -22553.783} C_VEL
LIN {X 0,Y 178.488,Z 297.877,A -85,B 0,C 180,E1 -22556.547,E2 -22556.547} C_VEL
LIN {X 0,Y 178.524,Z 297.871,A -85,B 0,C 180,E1 -22560.007,E2 -22560.007} C_VEL
LIN {X 0,Y 178.537,Z 297.868,A -85,B 0,C 180,E1 -22564.876,E2 -22564.876} C_VEL
LIN {X 0,Y 178.626,Z 297.859,A -85,B 0,C 180,E1 -22570.784,E2 -22570.784} C_VEL
LIN {X 0,Y 178.662,Z 297.854,A -85,B 0,C 180,E1 -22576.348,E2 -22576.348} C_VEL
LIN {X 0,Y 178.909,Z 297.822,A -85,B 0,C 180,E1 -22580.96,E2 -22580.96} C_VEL
LIN {X 0,Y 179.147,Z 297.795,A -85,B 0,C 180,E1 -22587.752,E2 -22587.752} C_VEL
LIN {X 0,Y 179.368,Z 297.765,A -85,B 0,C 180,E1 -22590,E2 -22590} C_VEL
LIN {X 0,Y 178.861,Z 297.829,A -85,B 0,C 180,E1 -22594.507,E2 -22594.507} C_VEL
LIN {X 0,Y 178.911,Z 297.82,A -85,B 0,C 180,E1 -22599.04,E2 -22599.04} C_VEL
LIN {X 0,Y 178.668,Z 297.856,A -85,B 0,C 180,E1 -22603.652,E2 -22603.652} C_VEL
LIN {X 0,Y 178.683,Z 297.848,A -85,B 0,C 180,E1 -22608.34,E2 -22608.34} C_VEL
LIN {X 0,Y 178.534,Z 297.871,A -85,B 0,C 180,E1 -22613.182,E2 -22613.182} C_VEL
LIN {X 0,Y 178.489,Z 297.874,A -85,B 0,C 180,E1 -22618.197,E2 -22618.197} C_VEL
LIN {X 0,Y 178.48,Z 297.877,A -85,B 0,C 180,E1 -22620.791,E2 -22620.791} C_VEL
LIN {X 0,Y 178.486,Z 297.871,A -85,B 0,C 180,E1 -22624.218,E2 -22624.218} C_VEL
LIN {X 0,Y 178.389,Z 297.89,A -85,B 0,C 180,E1 -22629.076,E2 -22629.076} C_VEL
LIN {X 0,Y 178.396,Z 297.883,A -85,B 0,C 180,E1 -22632.046,E2 -22632.046} C_VEL
LIN {X 0,Y 178.395,Z 297.889,A -85,B 0,C 180,E1 -22635.164,E2 -22635.164} C_VEL
LIN {X 0,Y 178.405,Z 297.886,A -85,B 0,C 180,E1 -22638.459,E2 -22638.459} C_VEL
LIN {X 0,Y 178.425,Z 297.883,A -85,B 0,C 180,E1 -22643.783,E2 -22643.783} C_VEL
LIN {X 0,Y 178.488,Z 297.877,A -85,B 0,C 180,E1 -22646.546,E2 -22646.546} C_VEL
LIN {X 0,Y 178.524,Z 297.868,A -85,B 0,C 180,E1 -22650.007,E2 -22650.007} C_VEL
LIN {X 0,Y 178.537,Z 297.869,A -85,B 0,C 180,E1 -22654.875,E2 -22654.875} C_VEL
LIN {X 0,Y 178.627,Z 297.859,A -85,B 0,C 180,E1 -22660.783,E2 -22660.783} C_VEL
LIN {X 0,Y 178.662,Z 297.852,A -85,B 0,C 180,E1 -22666.348,E2 -22666.348} C_VEL
LIN {X 0,Y 178.909,Z 297.822,A -85,B 0,C 180,E1 -22670.959,E2 -22670.959} C_VEL
LIN {X 0,Y 179.15,Z 297.794,A -85,B 0,C 180,E1 -22677.751,E2 -22677.751} C_VEL
LIN {X 0,Y 179.366,Z 297.766,A -85,B 0,C 180,E1 -22679.999,E2 -22679.999} C_VEL
LIN {X 0,Y 178.863,Z 297.829,A -85,B 0,C 180,E1 -22684.507,E2 -22684.507} C_VEL
LIN {X 0,Y 178.909,Z 297.821,A -85,B 0,C 180,E1 -22689.04,E2 -22689.04} C_VEL
LIN {X 0,Y 178.661,Z 297.856,A -85,B 0,C 180,E1 -22693.651,E2 -22693.651} C_VEL
LIN {X 0,Y 178.625,Z 297.857,A -85,B 0,C 180,E1 -22699.215,E2 -22699.215} C_VEL
LIN {X 0,Y 178.651,Z 297.892,A -85,B 0,C 180,E1 -22704.051,E2 -22704.051} C_VEL
LIN {X 0,Y 179.193,Z 302.335,A -85,B 0,C 180,E1 -22710.362,E2 -22710.362} C_VEL
LIN {X 0,Y 179.943,Z 306.431,A -85,B 0,C 180,E1 -22715.863,E2 -22715.863} C_VEL
LIN {X 0,Y 180.446,Z 308.749,A -85,B 0,C 180,E1 -22718.834,E2 -22718.834} C_VEL
LIN {X 0,Y 181.282,Z 312.258,A -85,B 0,C 180,E1 -22723.026,E2 -22723.026} C_VEL
LIN {X 0,Y 184.96,Z 325.768,A -85,B 0,C 180,E1 -22724.953,E2 -22724.953} C_VEL
LIN {X 0,Y 187.609,Z 342.312,A -85,B 0,C 180,E1 -22727.363,E2 -22727.363} C_VEL
LIN {X 0,Y 189.892,Z 359.019,A -85,B 0,C 180,E1 -22730.163,E2 -22730.163} C_VEL
LIN {X 0,Y 191.733,Z 373.164,A -85,B 0,C 180,E1 -22732.866,E2 -22732.866} C_VEL
LIN {X 0,Y 193.298,Z 386.311,A -85,B 0,C 180,E1 -22735.698,E2 -22735.698} C_VEL
LIN {X 0,Y 193.404,Z 387.808,A -85,B 0,C 180,E1 -22736.033,E2 -22736.033} C_VEL
LIN {X 0,Y 189.883,Z 399.767,A -85,B 0,C 180,E1 -22738.79,E2 -22738.79} C_VEL
LIN {X 0,Y 186.496,Z 410.928,A -85,B 0,C 180,E1 -22741.897,E2 -22741.897} C_VEL
LIN {X 0,Y 183.284,Z 422.06,A -85,B 0,C 180,E1 -22745.656,E2 -22745.656} C_VEL
LIN {X 0,Y 180.731,Z 431.395,A -85,B 0,C 180,E1 -22749.514,E2 -22749.514} C_VEL
LIN {X 0,Y 178.687,Z 440.273,A -85,B 0,C 180,E1 -22754.019,E2 -22754.019} C_VEL
LIN {X 0,Y 177.481,Z 447.447,A -85,B 0,C 180,E1 -22758.58,E2 -22758.58} C_VEL
LIN {X 0,Y 177.027,Z 453.086,A -85,B 0,C 180,E1 -22763.16,E2 -22763.16} C_VEL
LIN {X 0,Y 176.937,Z 455.36,A -85,B 0,C 180,E1 -22765.443,E2 -22765.443} C_VEL
LIN {X 0,Y 176.879,Z 458.886,A -85,B 0,C 180,E1 -22770,E2 -22770} C_VEL
LIN {X 0,Y 176.564,Z 461.125,A -85,B 0,C 180,E1 -22774.566,E2 -22774.566} C_VEL
LIN {X 0,Y 176.491,Z 462.207,A -85,B 0,C 180,E1 -22779.165,E2 -22779.165} C_VEL
LIN {X 0,Y 177.251,Z 462.447,A -85,B 0,C 180,E1 -22783.763,E2 -22783.763} C_VEL
LIN {X 0,Y 177.955,Z 462.249,A -85,B 0,C 180,E1 -22785.691,E2 -22785.691} C_VEL
LIN {X 0,Y 178.162,Z 461.981,A -85,B 0,C 180,E1 -22787.587,E2 -22787.587} C_VEL
LIN {X 0,Y 177.116,Z 461.245,A -85,B 0,C 180,E1 -22790.756,E2 -22790.756} C_VEL
LIN {X 0,Y 176.554,Z 460.41,A -85,B 0,C 180,E1 -22793.308,E2 -22793.308} C_VEL
LIN {X 0,Y 177.172,Z 459.644,A -85,B 0,C 180,E1 -22795.194,E2 -22795.194} C_VEL
LIN {X 0,Y 177.687,Z 459.365,A -85,B 0,C 180,E1 -22795.801,E2 -22795.801} C_VEL
LIN {X 0,Y 185.533,Z 455.891,A -85,B 0,C 180,E1 -22802.027,E2 -22802.027} C_VEL
LIN {X 0,Y 192.201,Z 452.795,A -85,B 0,C 180,E1 -22805.807,E2 -22805.807} C_VEL
LIN {X 0,Y 204.296,Z 447.102,A -85,B 0,C 180,E1 -22810.816,E2 -22810.816} C_VEL
LIN {X 0,Y 218.43,Z 440.164,A -85,B 0,C 180,E1 -22815.061,E2 -22815.061} C_VEL
LIN {X 0,Y 205.278,Z 444.574,A -85,B 0,C 180,E1 -22819.422,E2 -22819.422} C_VEL
LIN {X 0,Y 197.32,Z 446.756,A -85,B 0,C 180,E1 -22822.736,E2 -22822.736} C_VEL
LIN {X 0,Y 187.138,Z 448.745,A -85,B 0,C 180,E1 -22828.28,E2 -22828.28} C_VEL
LIN {X 0,Y 181.548,Z 449.068,A -85,B 0,C 180,E1 -22832.32,E2 -22832.32} C_VEL
LIN {X 0,Y 177.028,Z 448.617,A -85,B 0,C 180,E1 -22836.61,E2 -22836.61} C_VEL
LIN {X 0,Y 173.577,Z 447.21,A -85,B 0,C 180,E1 -22841.101,E2 -22841.101} C_VEL
LIN {X 0,Y 171.249,Z 444.893,A -85,B 0,C 180,E1 -22845.746,E2 -22845.746} C_VEL
LIN {X 0,Y 169.918,Z 441.606,A -85,B 0,C 180,E1 -22850.478,E2 -22850.478} C_VEL
LIN {X 0,Y 169.368,Z 436.513,A -85,B 0,C 180,E1 -22855.908,E2 -22855.908} C_VEL
LIN {X 0,Y 169.478,Z 431.601,A -85,B 0,C 180,E1 -22860.001,E2 -22860.001} C_VEL
LIN {X 0,Y 169.948,Z 424.645,A -85,B 0,C 180,E1 -22864.745,E2 -22864.745} C_VEL
LIN {X 0,Y 170.876,Z 416.105,A -85,B 0,C 180,E1 -22869.47,E2 -22869.47} C_VEL
LIN {X 0,Y 172.566,Z 405.835,A -85,B 0,C 180,E1 -22874.145,E2 -22874.145} C_VEL
LIN {X 0,Y 174.787,Z 395.053,A -85,B 0,C 180,E1 -22878.158,E2 -22878.158} C_VEL
LIN {X 0,Y 177.605,Z 382.338,A -85,B 0,C 180,E1 -22882.082,E2 -22882.082} C_VEL
LIN {X 0,Y 180.849,Z 368.346,A -85,B 0,C 180,E1 -22885.616,E2 -22885.616} C_VEL
LIN {X 0,Y 183.95,Z 353.932,A -85,B 0,C 180,E1 -22888.602,E2 -22888.602} C_VEL
LIN {X 0,Y 185.335,Z 346.775,A -85,B 0,C 180,E1 -22889.879,E2 -22889.879} C_VEL
LIN {X 0,Y 182.349,Z 332.573,A -85,B 0,C 180,E1 -22892.656,E2 -22892.656} C_VEL
LIN {X 0,Y 177.937,Z 317.958,A -85,B 0,C 180,E1 -22895.338,E2 -22895.338} C_VEL
LIN {X 0,Y 173.13,Z 303.971,A -85,B 0,C 180,E1 -22897.75,E2 -22897.75} C_VEL
LIN {X 0,Y 171.347,Z 298.771,A -85,B 0,C 180,E1 -22898.646,E2 -22898.646} C_VEL
LIN {X 0,Y 171.322,Z 298.771,A -85,B 0,C 180,E1 -22904.218,E2 -22904.218} C_VEL
LIN {X 0,Y 171.337,Z 298.769,A -85,B 0,C 180,E1 -22908.982,E2 -22908.982} C_VEL
LIN {X 0,Y 171.39,Z 298.76,A -85,B 0,C 180,E1 -22912.041,E2 -22912.041} C_VEL
LIN {X 0,Y 171.4,Z 298.76,A -85,B 0,C 180,E1 -22915.093,E2 -22915.093} C_VEL
LIN {X 0,Y 171.451,Z 298.753,A -85,B 0,C 180,E1 -22920.535,E2 -22920.535} C_VEL
LIN {X 0,Y 171.461,Z 298.748,A -85,B 0,C 180,E1 -22925.802,E2 -22925.802} C_VEL
LIN {X 0,Y 171.582,Z 298.736,A -85,B 0,C 180,E1 -22930.872,E2 -22930.872} C_VEL
LIN {X 0,Y 171.58,Z 298.733,A -85,B 0,C 180,E1 -22935.773,E2 -22935.773} C_VEL
LIN {X 0,Y 171.847,Z 298.702,A -85,B 0,C 180,E1 -22940.585,E2 -22940.585} C_VEL
LIN {X 0,Y 171.802,Z 298.707,A -85,B 0,C 180,E1 -22945.307,E2 -22945.307} C_VEL
LIN {X 0,Y 172.331,Z 298.641,A -85,B 0,C 180,E1 -22950,E2 -22950} C_VEL
LIN {X 0,Y 171.809,Z 298.707,A -85,B 0,C 180,E1 -22954.693,E2 -22954.693} C_VEL
LIN {X 0,Y 171.849,Z 298.7,A -85,B 0,C 180,E1 -22959.415,E2 -22959.415} C_VEL
LIN {X 0,Y 171.597,Z 298.734,A -85,B 0,C 180,E1 -22964.226,E2 -22964.226} C_VEL
LIN {X 0,Y 171.614,Z 298.729,A -85,B 0,C 180,E1 -22969.125,E2 -22969.125} C_VEL
LIN {X 0,Y 171.472,Z 298.746,A -85,B 0,C 180,E1 -22975.616,E2 -22975.616} C_VEL
LIN {X 0,Y 171.443,Z 298.753,A -85,B 0,C 180,E1 -22980.586,E2 -22980.586} C_VEL
LIN {X 0,Y 171.394,Z 298.756,A -85,B 0,C 180,E1 -22985.035,E2 -22985.035} C_VEL
LIN {X 0,Y 171.345,Z 298.767,A -85,B 0,C 180,E1 -22988.801,E2 -22988.801} C_VEL
LIN {X 0,Y 171.321,Z 298.766,A -85,B 0,C 180,E1 -22994.218,E2 -22994.218} C_VEL
LIN {X 0,Y 171.338,Z 298.766,A -85,B 0,C 180,E1 -22998.981,E2 -22998.981} C_VEL
LIN {X 0,Y 171.39,Z 298.757,A -85,B 0,C 180,E1 -23002.041,E2 -23002.041} C_VEL
LIN {X 0,Y 171.401,Z 298.76,A -85,B 0,C 180,E1 -23005.092,E2 -23005.092} C_VEL
LIN {X 0,Y 171.451,Z 298.751,A -85,B 0,C 180,E1 -23010.534,E2 -23010.534} C_VEL
LIN {X 0,Y 171.461,Z 298.749,A -85,B 0,C 180,E1 -23015.801,E2 -23015.801} C_VEL
LIN {X 0,Y 171.583,Z 298.737,A -85,B 0,C 180,E1 -23020.871,E2 -23020.871} C_VEL
LIN {X 0,Y 171.58,Z 298.732,A -85,B 0,C 180,E1 -23025.772,E2 -23025.772} C_VEL
LIN {X 0,Y 171.847,Z 298.703,A -85,B 0,C 180,E1 -23030.584,E2 -23030.584} C_VEL
LIN {X 0,Y 171.807,Z 298.706,A -85,B 0,C 180,E1 -23035.307,E2 -23035.307} C_VEL
LIN {X 0,Y 172.33,Z 298.643,A -85,B 0,C 180,E1 -23039.999,E2 -23039.999} C_VEL
LIN {X 0,Y 171.811,Z 298.707,A -85,B 0,C 180,E1 -23044.692,E2 -23044.692} C_VEL
LIN {X 0,Y 171.847,Z 298.702,A -85,B 0,C 180,E1 -23049.415,E2 -23049.415} C_VEL
LIN {X 0,Y 171.579,Z 298.737,A -85,B 0,C 180,E1 -23054.226,E2 -23054.226} C_VEL
LIN {X 0,Y 171.545,Z 298.74,A -85,B 0,C 180,E1 -23059.56,E2 -23059.56} C_VEL
LIN {X 0,Y 171.642,Z 298.911,A -85,B 0,C 180,E1 -23064.17,E2 -23064.17} C_VEL
LIN {X 0,Y 172.204,Z 303.591,A -85,B 0,C 180,E1 -23071.012,E2 -23071.012} C_VEL
LIN {X 0,Y 172.852,Z 306.894,A -85,B 0,C 180,E1 -23075.592,E2 -23075.592} C_VEL
LIN {X 0,Y 173.934,Z 311.704,A -85,B 0,C 180,E1 -23081.909,E2 -23081.909} C_VEL
LIN {X 0,Y 178.029,Z 326.097,A -85,B 0,C 180,E1 -23084.096,E2 -23084.096} C_VEL
LIN {X 0,Y 180.122,Z 338.58,A -85,B 0,C 180,E1 -23085.982,E2 -23085.982} C_VEL
LIN {X 0,Y 182.428,Z 355.398,A -85,B 0,C 180,E1 -23088.842,E2 -23088.842} C_VEL
LIN {X 0,Y 184.327,Z 370.218,A -85,B 0,C 180,E1 -23091.715,E2 -23091.715} C_VEL
LIN {X 0,Y 185.927,Z 384.242,A -85,B 0,C 180,E1 -23094.799,E2 -23094.799} C_VEL
LIN {X 0,Y 186.307,Z 387.369,A -85,B 0,C 180,E1 -23095.539,E2 -23095.539} C_VEL
LIN {X 0,Y 183.515,Z 397.33,A -85,B 0,C 180,E1 -23097.902,E2 -23097.902} C_VEL
LIN {X 0,Y 179.705,Z 409.591,A -85,B 0,C 180,E1 -23101.374,E2 -23101.374} C_VEL
LIN {X 0,Y 176.403,Z 420.784,A -85,B 0,C 180,E1 -23105.271,E2 -23105.271} C_VEL
LIN {X 0,Y 173.778,Z 430.205,A -85,B 0,C 180,E1 -23109.275,E2 -23109.275} C_VEL
LIN {X 0,Y 171.691,Z 439.137,A -85,B 0,C 180,E1 -23113.96,E2 -23113.96} C_VEL
LIN {X 0,Y 170.574,Z 445.561,A -85,B 0,C 180,E1 -23118.111,E2 -23118.111} C_VEL
LIN {X 0,Y 170.071,Z 451.457,A -85,B 0,C 180,E1 -23122.878,E2 -23122.878} C_VEL
LIN {X 0,Y 169.896,Z 454.897,A -85,B 0,C 180,E1 -23126.442,E2 -23126.442} C_VEL
LIN {X 0,Y 169.889,Z 457.605,A -85,B 0,C 180,E1 -23130,E2 -23130} C_VEL
LIN {X 0,Y 169.56,Z 459.973,A -85,B 0,C 180,E1 -23134.755,E2 -23134.755} C_VEL
LIN {X 0,Y 169.492,Z 461.319,A -85,B 0,C 180,E1 -23139.547,E2 -23139.547} C_VEL
LIN {X 0,Y 171.253,Z 461.62,A -85,B 0,C 180,E1 -23146.695,E2 -23146.695} C_VEL
LIN {X 0,Y 174.027,Z 460.731,A -85,B 0,C 180,E1 -23151.746,E2 -23151.746} C_VEL
LIN {X 0,Y 177.687,Z 459.365,A -85,B 0,C 180,E1 -23155.801,E2 -23155.801} C_VEL
LIN {X 0,Y 178.963,Z 458.544,A -85,B 0,C 180,E1 -23157.636,E2 -23157.636} C_VEL
LIN {X 0,Y 180.807,Z 456.054,A -85,B 0,C 180,E1 -23163.233,E2 -23163.233} C_VEL
LIN {X 0,Y 182.58,Z 455.004,A -85,B 0,C 180,E1 -23164.972,E2 -23164.972} C_VEL
LIN {X 0,Y 183.461,Z 454.613,A -85,B 0,C 180,E1 -23165.507,E2 -23165.507} C_VEL
LIN {X 0,Y 194.654,Z 450.082,A -85,B 0,C 180,E1 -23170.534,E2 -23170.534} C_VEL
LIN {X 0,Y 208.553,Z 444.12,A -85,B 0,C 180,E1 -23175.047,E2 -23175.047} C_VEL
LIN {X 0,Y 204.601,Z 445.196,A -85,B 0,C 180,E1 -23176.608,E2 -23176.608} C_VEL
LIN {X 0,Y 191.833,Z 448.245,A -85,B 0,C 180,E1 -23181.479,E2 -23181.479} C_VEL
LIN {X 0,Y 181.168,Z 449.729,A -85,B 0,C 180,E1 -23187.106,E2 -23187.106} C_VEL
LIN {X 0,Y 175.285,Z 449.831,A -85,B 0,C 180,E1 -23191.241,E2 -23191.241} C_VEL
LIN {X 0,Y 170.521,Z 449.047,A -85,B 0,C 180,E1 -23195.661,E2 -23195.661} C_VEL
LIN {X 0,Y 166.837,Z 447.454,A -85,B 0,C 180,E1 -23200.306,E2 -23200.306} C_VEL
LIN {X 0,Y 164.34,Z 444.886,A -85,B 0,C 180,E1 -23205.133,E2 -23205.133} C_VEL
LIN {X 0,Y 162.69,Z 440.33,A -85,B 0,C 180,E1 -23211.304,E2 -23211.304} C_VEL
LIN {X 0,Y 162.301,Z 435.726,A -85,B 0,C 180,E1 -23216.013,E2 -23216.013} C_VEL
LIN {X 0,Y 162.416,Z 431.002,A -85,B 0,C 180,E1 -23220.001,E2 -23220.001} C_VEL
LIN {X 0,Y 162.911,Z 423.825,A -85,B 0,C 180,E1 -23224.95,E2 -23224.95} C_VEL
LIN {X 0,Y 163.908,Z 415.051,A -85,B 0,C 180,E1 -23229.876,E2 -23229.876} C_VEL
LIN {X 0,Y 165.711,Z 404.419,A -85,B 0,C 180,E1 -23234.743,E2 -23234.743} C_VEL
LIN {X 0,Y 168.048,Z 393.43,A -85,B 0,C 180,E1 -23238.913,E2 -23238.913} C_VEL
LIN {X 0,Y 170.796,Z 381.346,A -85,B 0,C 180,E1 -23242.692,E2 -23242.692} C_VEL
LIN {X 0,Y 174.15,Z 367.104,A -85,B 0,C 180,E1 -23246.355,E2 -23246.355} C_VEL
LIN {X 0,Y 177.297,Z 352.911,A -85,B 0,C 180,E1 -23249.357,E2 -23249.357} C_VEL
LIN {X 0,Y 178.279,Z 348.457,A -85,B 0,C 180,E1 -23250.179,E2 -23250.179} C_VEL
LIN {X 0,Y 177.491,Z 343.019,A -85,B 0,C 180,E1 -23251.303,E2 -23251.303} C_VEL
LIN {X 0,Y 174.909,Z 332.019,A -85,B 0,C 180,E1 -23253.514,E2 -23253.514} C_VEL
LIN {X 0,Y 170.115,Z 316.367,A -85,B 0,C 180,E1 -23256.527,E2 -23256.527} C_VEL
LIN {X 0,Y 165.203,Z 302.436,A -85,B 0,C 180,E1 -23259.069,E2 -23259.069} C_VEL
LIN {X 0,Y 164.269,Z 299.654,A -85,B 0,C 180,E1 -23259.576,E2 -23259.576} C_VEL
LIN {X 0,Y 164.282,Z 299.65,A -85,B 0,C 180,E1 -23263.342,E2 -23263.342} C_VEL
LIN {X 0,Y 164.266,Z 299.649,A -85,B 0,C 180,E1 -23266.799,E2 -23266.799} C_VEL
LIN {X 0,Y 164.297,Z 299.644,A -85,B 0,C 180,E1 -23270.352,E2 -23270.352} C_VEL
LIN {X 0,Y 164.332,Z 299.64,A -85,B 0,C 180,E1 -23274.349,E2 -23274.349} C_VEL
LIN {X 0,Y 164.392,Z 299.632,A -85,B 0,C 180,E1 -23279.135,E2 -23279.135} C_VEL
LIN {X 0,Y 164.419,Z 299.627,A -85,B 0,C 180,E1 -23284.694,E2 -23284.694} C_VEL
LIN {X 0,Y 164.488,Z 299.62,A -85,B 0,C 180,E1 -23290.051,E2 -23290.051} C_VEL
LIN {X 0,Y 164.527,Z 299.61,A -85,B 0,C 180,E1 -23295.149,E2 -23295.149} C_VEL
LIN {X 0,Y 164.768,Z 299.586,A -85,B 0,C 180,E1 -23300.176,E2 -23300.176} C_VEL
LIN {X 0,Y 164.826,Z 299.573,A -85,B 0,C 180,E1 -23302.651,E2 -23302.651} C_VEL
LIN {X 0,Y 165.042,Z 299.551,A -85,B 0,C 180,E1 -23307.559,E2 -23307.559} C_VEL
LIN {X 0,Y 165.294,Z 299.517,A -85,B 0,C 180,E1 -23310,E2 -23310} C_VEL
LIN {X 0,Y 164.758,Z 299.586,A -85,B 0,C 180,E1 -23314.894,E2 -23314.894} C_VEL
LIN {X 0,Y 164.829,Z 299.577,A -85,B 0,C 180,E1 -23317.349,E2 -23317.349} C_VEL
LIN {X 0,Y 164.621,Z 299.603,A -85,B 0,C 180,E1 -23322.325,E2 -23322.325} C_VEL
LIN {X 0,Y 164.528,Z 299.612,A -85,B 0,C 180,E1 -23327.399,E2 -23327.399} C_VEL
LIN {X 0,Y 164.523,Z 299.615,A -85,B 0,C 180,E1 -23329.983,E2 -23329.983} C_VEL
LIN {X 0,Y 164.396,Z 299.627,A -85,B 0,C 180,E1 -23336.134,E2 -23336.134} C_VEL
LIN {X 0,Y 164.377,Z 299.635,A -85,B 0,C 180,E1 -23341.227,E2 -23341.227} C_VEL
LIN {X 0,Y 164.282,Z 299.645,A -85,B 0,C 180,E1 -23346.793,E2 -23346.793} C_VEL
LIN {X 0,Y 164.288,Z 299.644,A -85,B 0,C 180,E1 -23349.918,E2 -23349.918} C_VEL
LIN {X 0,Y 164.282,Z 299.644,A -85,B 0,C 180,E1 -23353.342,E2 -23353.342} C_VEL
LIN {X 0,Y 164.266,Z 299.649,A -85,B 0,C 180,E1 -23356.799,E2 -23356.799} C_VEL
LIN {X 0,Y 164.298,Z 299.64,A -85,B 0,C 180,E1 -23360.352,E2 -23360.352} C_VEL
LIN {X 0,Y 164.333,Z 299.639,A -85,B 0,C 180,E1 -23364.349,E2 -23364.349} C_VEL
LIN {X 0,Y 164.392,Z 299.628,A -85,B 0,C 180,E1 -23369.134,E2 -23369.134} C_VEL
LIN {X 0,Y 164.419,Z 299.628,A -85,B 0,C 180,E1 -23374.694,E2 -23374.694} C_VEL
LIN {X 0,Y 164.488,Z 299.62,A -85,B 0,C 180,E1 -23380.051,E2 -23380.051} C_VEL
LIN {X 0,Y 164.527,Z 299.61,A -85,B 0,C 180,E1 -23385.149,E2 -23385.149} C_VEL
LIN {X 0,Y 164.768,Z 299.587,A -85,B 0,C 180,E1 -23390.176,E2 -23390.176} C_VEL
LIN {X 0,Y 164.826,Z 299.574,A -85,B 0,C 180,E1 -23392.65,E2 -23392.65} C_VEL
LIN {X 0,Y 165.045,Z 299.551,A -85,B 0,C 180,E1 -23397.559,E2 -23397.559} C_VEL
LIN {X 0,Y 165.293,Z 299.519,A -85,B 0,C 180,E1 -23399.999,E2 -23399.999} C_VEL
LIN {X 0,Y 164.76,Z 299.585,A -85,B 0,C 180,E1 -23404.893,E2 -23404.893} C_VEL
LIN {X 0,Y 164.827,Z 299.578,A -85,B 0,C 180,E1 -23407.349,E2 -23407.349} C_VEL
LIN {X 0,Y 164.704,Z 299.589,A -85,B 0,C 180,E1 -23411.06,E2 -23411.06} C_VEL
LIN {X 0,Y 164.486,Z 299.619,A -85,B 0,C 180,E1 -23417.402,E2 -23417.402} C_VEL
LIN {X 0,Y 164.471,Z 299.624,A -85,B 0,C 180,E1 -23422.617,E2 -23422.617} C_VEL
LIN {X 0,Y 164.553,Z 299.657,A -85,B 0,C 180,E1 -23423.937,E2 -23423.937} C_VEL
LIN {X 0,Y 164.793,Z 302.295,A -85,B 0,C 180,E1 -23427.977,E2 -23427.977} C_VEL
LIN {X 0,Y 165.217,Z 304.798,A -85,B 0,C 180,E1 -23431.705,E2 -23431.705} C_VEL
LIN {X 0,Y 165.89,Z 308.092,A -85,B 0,C 180,E1 -23436.395,E2 -23436.395} C_VEL
LIN {X 0,Y 166.623,Z 311.434,A -85,B 0,C 180,E1 -23440.777,E2 -23440.777} C_VEL
LIN {X 0,Y 170.945,Z 325.881,A -85,B 0,C 180,E1 -23443.117,E2 -23443.117} C_VEL
LIN {X 0,Y 172.869,Z 335.947,A -85,B 0,C 180,E1 -23444.742,E2 -23444.742} C_VEL
LIN {X 0,Y 174.996,Z 352.26,A -85,B 0,C 180,E1 -23447.555,E2 -23447.555} C_VEL
LIN {X 0,Y 176.901,Z 367.351,A -85,B 0,C 180,E1 -23450.531,E2 -23450.531} C_VEL
LIN {X 0,Y 178.569,Z 381.975,A -85,B 0,C 180,E1 -23453.817,E2 -23453.817} C_VEL
LIN {X 0,Y 179.176,Z 387.239,A -85,B 0,C 180,E1 -23455.112,E2 -23455.112} C_VEL
LIN {X 0,Y 177.88,Z 392.621,A -85,B 0,C 180,E1 -23456.417,E2 -23456.417} C_VEL
LIN {X 0,Y 174.084,Z 404.572,A -85,B 0,C 180,E1 -23459.692,E2 -23459.692} C_VEL
LIN {X 0,Y 170.394,Z 416.403,A -85,B 0,C 180,E1 -23463.679,E2 -23463.679} C_VEL
LIN {X 0,Y 167.536,Z 426.386,A -85,B 0,C 180,E1 -23467.818,E2 -23467.818} C_VEL
LIN {X 0,Y 165.338,Z 434.754,A -85,B 0,C 180,E1 -23472.051,E2 -23472.051} C_VEL
LIN {X 0,Y 163.978,Z 441.787,A -85,B 0,C 180,E1 -23476.365,E2 -23476.365} C_VEL
LIN {X 0,Y 163.173,Z 448.459,A -85,B 0,C 180,E1 -23481.454,E2 -23481.454} C_VEL
LIN {X 0,Y 163.014,Z 452.239,A -85,B 0,C 180,E1 -23485.053,E2 -23485.053} C_VEL
LIN {X 0,Y 162.919,Z 456.176,A -85,B 0,C 180,E1 -23490,E2 -23490} C_VEL
LIN {X 0,Y 162.557,Z 458.797,A -85,B 0,C 180,E1 -23494.96,E2 -23494.96} C_VEL
LIN {X 0,Y 162.508,Z 460.27,A -85,B 0,C 180,E1 -23499.962,E2 -23499.962} C_VEL
LIN {X 0,Y 163.434,Z 460.927,A -85,B 0,C 180,E1 -23504.952,E2 -23504.952} C_VEL
LIN {X 0,Y 167.187,Z 460.384,A -85,B 0,C 180,E1 -23512.362,E2 -23512.362} C_VEL
LIN {X 0,Y 173.731,Z 458.33,A -85,B 0,C 180,E1 -23519.041,E2 -23519.041} C_VEL
LIN {X 0,Y 183.461,Z 454.613,A -85,B 0,C 180,E1 -23525.507,E2 -23525.507} C_VEL
LIN {X 0,Y 185.895,Z 453.48,A -85,B 0,C 180,E1 -23527.143,E2 -23527.143} C_VEL
LIN {X 0,Y 191.515,Z 450.349,A -85,B 0,C 180,E1 -23532.195,E2 -23532.195} C_VEL
LIN {X 0,Y 194.435,Z 449.067,A -85,B 0,C 180,E1 -23533.66,E2 -23533.66} C_VEL
LIN {X 0,Y 195.656,Z 448.586,A -85,B 0,C 180,E1 -23534.087,E2 -23534.087} C_VEL
LIN {X 0,Y 198.699,Z 447.427,A -85,B 0,C 180,E1 -23535.024,E2 -23535.024} C_VEL
LIN {X 0,Y 195.07,Z 448.077,A -85,B 0,C 180,E1 -23536.802,E2 -23536.802} C_VEL
LIN {X 0,Y 186.441,Z 449.617,A -85,B 0,C 180,E1 -23540.147,E2 -23540.147} C_VEL
LIN {X 0,Y 175.286,Z 450.685,A -85,B 0,C 180,E1 -23545.853,E2 -23545.853} C_VEL
LIN {X 0,Y 166.424,Z 450.063,A -85,B 0,C 180,E1 -23552.321,E2 -23552.321} C_VEL
LIN {X 0,Y 161.93,Z 448.616,A -85,B 0,C 180,E1 -23557.008,E2 -23557.008} C_VEL
LIN {X 0,Y 158.593,Z 446.302,A -85,B 0,C 180,E1 -23561.929,E2 -23561.929} C_VEL
LIN {X 0,Y 156.552,Z 443.079,A -85,B 0,C 180,E1 -23567.029,E2 -23567.029} C_VEL
LIN {X 0,Y 155.351,Z 437.588,A -85,B 0,C 180,E1 -23573.508,E2 -23573.508} C_VEL
LIN {X 0,Y 155.31,Z 431.899,A -85,B 0,C 180,E1 -23578.704,E2 -23578.704} C_VEL
LIN {X 0,Y 155.688,Z 424.842,A -85,B 0,C 180,E1 -23583.883,E2 -23583.883} C_VEL
LIN {X 0,Y 156.449,Z 417.334,A -85,B 0,C 180,E1 -23588.427,E2 -23588.427} C_VEL
LIN {X 0,Y 157.748,Z 408.626,A -85,B 0,C 180,E1 -23592.872,E2 -23592.872} C_VEL
LIN {X 0,Y 159.855,Z 398.278,A -85,B 0,C 180,E1 -23597.264,E2 -23597.264} C_VEL
LIN {X 0,Y 162.566,Z 386.104,A -85,B 0,C 180,E1 -23601.56,E2 -23601.56} C_VEL
LIN {X 0,Y 165.492,Z 373.929,A -85,B 0,C 180,E1 -23605.131,E2 -23605.131} C_VEL
LIN {X 0,Y 168.307,Z 362.072,A -85,B 0,C 180,E1 -23608.02,E2 -23608.02} C_VEL
LIN {X 0,Y 171.339,Z 348.245,A -85,B 0,C 180,E1 -23610.845,E2 -23610.845} C_VEL
LIN {X 0,Y 168.661,Z 335.683,A -85,B 0,C 180,E1 -23613.551,E2 -23613.551} C_VEL
LIN {X 0,Y 164.119,Z 320.436,A -85,B 0,C 180,E1 -23616.691,E2 -23616.691} C_VEL
LIN {X 0,Y 159.625,Z 307.418,A -85,B 0,C 180,E1 -23619.203,E2 -23619.203} C_VEL
LIN {X 0,Y 157.195,Z 300.535,A -85,B 0,C 180,E1 -23620.531,E2 -23620.531} C_VEL
LIN {X 0,Y 157.18,Z 300.533,A -85,B 0,C 180,E1 -23625.678,E2 -23625.678} C_VEL
LIN {X 0,Y 157.208,Z 300.528,A -85,B 0,C 180,E1 -23631.254,E2 -23631.254} C_VEL
LIN {X 0,Y 157.281,Z 300.519,A -85,B 0,C 180,E1 -23634.486,E2 -23634.486} C_VEL
LIN {X 0,Y 157.295,Z 300.516,A -85,B 0,C 180,E1 -23638.097,E2 -23638.097} C_VEL
LIN {X 0,Y 157.324,Z 300.512,A -85,B 0,C 180,E1 -23643.466,E2 -23643.466} C_VEL
LIN {X 0,Y 157.397,Z 300.503,A -85,B 0,C 180,E1 -23649.668,E2 -23649.668} C_VEL
LIN {X 0,Y 157.457,Z 300.492,A -85,B 0,C 180,E1 -23654.466,E2 -23654.466} C_VEL
LIN {X 0,Y 157.691,Z 300.467,A -85,B 0,C 180,E1 -23659.731,E2 -23659.731} C_VEL
LIN {X 0,Y 157.764,Z 300.453,A -85,B 0,C 180,E1 -23662.32,E2 -23662.32} C_VEL
LIN {X 0,Y 158.256,Z 300.394,A -85,B 0,C 180,E1 -23670,E2 -23670} C_VEL
LIN {X 0,Y 157.766,Z 300.457,A -85,B 0,C 180,E1 -23677.68,E2 -23677.68} C_VEL
LIN {X 0,Y 157.641,Z 300.47,A -85,B 0,C 180,E1 -23681.238,E2 -23681.238} C_VEL
LIN {X 0,Y 157.483,Z 300.493,A -85,B 0,C 180,E1 -23685.531,E2 -23685.531} C_VEL
LIN {X 0,Y 157.419,Z 300.5,A -85,B 0,C 180,E1 -23690.926,E2 -23690.926} C_VEL
LIN {X 0,Y 157.317,Z 300.508,A -85,B 0,C 180,E1 -23696.684,E2 -23696.684} C_VEL
LIN {X 0,Y 157.277,Z 300.516,A -85,B 0,C 180,E1 -23702.427,E2 -23702.427} C_VEL
LIN {X 0,Y 157.261,Z 300.518,A -85,B 0,C 180,E1 -23706.444,E2 -23706.444} C_VEL
LIN {X 0,Y 157.192,Z 300.524,A -85,B 0,C 180,E1 -23712.117,E2 -23712.117} C_VEL
LIN {X 0,Y 157.195,Z 300.527,A -85,B 0,C 180,E1 -23717.883,E2 -23717.883} C_VEL
LIN {X 0,Y 157.271,Z 300.518,A -85,B 0,C 180,E1 -23723.55,E2 -23723.55} C_VEL
LIN {X 0,Y 157.295,Z 300.513,A -85,B 0,C 180,E1 -23728.096,E2 -23728.096} C_VEL
LIN {X 0,Y 157.325,Z 300.512,A -85,B 0,C 180,E1 -23733.466,E2 -23733.466} C_VEL
LIN {X 0,Y 157.397,Z 300.502,A -85,B 0,C 180,E1 -23739.667,E2 -23739.667} C_VEL
LIN {X 0,Y 157.457,Z 300.492,A -85,B 0,C 180,E1 -23744.466,E2 -23744.466} C_VEL
LIN {X 0,Y 157.69,Z 300.467,A -85,B 0,C 180,E1 -23749.73,E2 -23749.73} C_VEL
LIN {X 0,Y 157.764,Z 300.455,A -85,B 0,C 180,E1 -23752.319,E2 -23752.319} C_VEL
LIN {X 0,Y 158.255,Z 300.395,A -85,B 0,C 180,E1 -23759.999,E2 -23759.999} C_VEL
LIN {X 0,Y 157.765,Z 300.458,A -85,B 0,C 180,E1 -23767.679,E2 -23767.679} C_VEL
LIN {X 0,Y 157.639,Z 300.469,A -85,B 0,C 180,E1 -23771.236,E2 -23771.236} C_VEL
LIN {X 0,Y 157.456,Z 300.497,A -85,B 0,C 180,E1 -23775.533,E2 -23775.533} C_VEL
LIN {X 0,Y 157.418,Z 300.502,A -85,B 0,C 180,E1 -23780.925,E2 -23780.925} C_VEL
LIN {X 0,Y 157.533,Z 300.586,A -85,B 0,C 180,E1 -23784.022,E2 -23784.022} C_VEL
LIN {X 0,Y 157.854,Z 303.932,A -85,B 0,C 180,E1 -23789.323,E2 -23789.323} C_VEL
LIN {X 0,Y 158.66,Z 307.805,A -85,B 0,C 180,E1 -23795.158,E2 -23795.158} C_VEL
LIN {X 0,Y 159.314,Z 310.924,A -85,B 0,C 180,E1 -23799.56,E2 -23799.56} C_VEL
LIN {X 0,Y 164.279,Z 327.46,A -85,B 0,C 180,E1 -23802.412,E2 -23802.412} C_VEL
LIN {X 0,Y 166.087,Z 336.697,A -85,B 0,C 180,E1 -23803.998,E2 -23803.998} C_VEL
LIN {X 0,Y 168.07,Z 352.554,A -85,B 0,C 180,E1 -23806.87,E2 -23806.87} C_VEL
LIN {X 0,Y 169.849,Z 367.42,A -85,B 0,C 180,E1 -23809.95,E2 -23809.95} C_VEL
LIN {X 0,Y 171.33,Z 380.968,A -85,B 0,C 180,E1 -23813.117,E2 -23813.117} C_VEL
LIN {X 0,Y 172.077,Z 387.426,A -85,B 0,C 180,E1 -23814.769,E2 -23814.769} C_VEL
LIN {X 0,Y 171.313,Z 390.91,A -85,B 0,C 180,E1 -23815.661,E2 -23815.661} C_VEL
LIN {X 0,Y 167.407,Z 402.959,A -85,B 0,C 180,E1 -23819.051,E2 -23819.051} C_VEL
LIN {X 0,Y 163.596,Z 414.907,A -85,B 0,C 180,E1 -23823.187,E2 -23823.187} C_VEL
LIN {X 0,Y 160.653,Z 424.973,A -85,B 0,C 180,E1 -23827.494,E2 -23827.494} C_VEL
LIN {X 0,Y 158.375,Z 433.43,A -85,B 0,C 180,E1 -23831.903,E2 -23831.903} C_VEL
LIN {X 0,Y 157.132,Z 439.637,A -85,B 0,C 180,E1 -23835.759,E2 -23835.759} C_VEL
LIN {X 0,Y 156.244,Z 446.599,A -85,B 0,C 180,E1 -23841.072,E2 -23841.072} C_VEL
LIN {X 0,Y 156.029,Z 451.696,A -85,B 0,C 180,E1 -23846.126,E2 -23846.126} C_VEL
LIN {X 0,Y 155.953,Z 454.715,A -85,B 0,C 180,E1 -23850,E2 -23850} C_VEL
LIN {X 0,Y 155.596,Z 457.473,A -85,B 0,C 180,E1 -23855.183,E2 -23855.183} C_VEL
LIN {X 0,Y 155.54,Z 459.188,A -85,B 0,C 180,E1 -23860.413,E2 -23860.413} C_VEL
LIN {X 0,Y 157.638,Z 460.144,A -85,B 0,C 180,E1 -23868.185,E2 -23868.185} C_VEL
LIN {X 0,Y 160.53,Z 459.832,A -85,B 0,C 180,E1 -23873.205,E2 -23873.205} C_VEL
LIN {X 0,Y 167.531,Z 458.16,A -85,B 0,C 180,E1 -23880.226,E2 -23880.226} C_VEL
LIN {X 0,Y 177.424,Z 455.035,A -85,B 0,C 180,E1 -23886.685,E2 -23886.685} C_VEL
LIN {X 0,Y 185.016,Z 452.431,A -85,B 0,C 180,E1 -23890.223,E2 -23890.223} C_VEL
LIN {X 0,Y 195.656,Z 448.586,A -85,B 0,C 180,E1 -23894.087,E2 -23894.087} C_VEL
LIN {X 0,Y 196.048,Z 448.365,A -85,B 0,C 180,E1 -23894.558,E2 -23894.558} C_VEL
LIN {X 0,Y 195.208,Z 448.415,A -85,B 0,C 180,E1 -23895.21,E2 -23895.21} C_VEL
LIN {X 0,Y 192.702,Z 448.884,A -85,B 0,C 180,E1 -23896.034,E2 -23896.034} C_VEL
LIN {X 0,Y 183.361,Z 450.654,A -85,B 0,C 180,E1 -23897.991,E2 -23897.991} C_VEL
LIN {X 0,Y 181.068,Z 450.93,A -85,B 0,C 180,E1 -23898.758,E2 -23898.758} C_VEL
LIN {X 0,Y 173.135,Z 451.479,A -85,B 0,C 180,E1 -23902.491,E2 -23902.491} C_VEL
LIN {X 0,Y 166.066,Z 451.374,A -85,B 0,C 180,E1 -23906.622,E2 -23906.622} C_VEL
LIN {X 0,Y 159.14,Z 450.241,A -85,B 0,C 180,E1 -23912.037,E2 -23912.037} C_VEL
LIN {X 0,Y 153.479,Z 447.647,A -85,B 0,C 180,E1 -23918.511,E2 -23918.511} C_VEL
LIN {X 0,Y 150.607,Z 444.618,A -85,B 0,C 180,E1 -23923.741,E2 -23923.741} C_VEL
LIN {X 0,Y 148.925,Z 440.671,A -85,B 0,C 180,E1 -23929.12,E2 -23929.12} C_VEL
LIN {X 0,Y 148.215,Z 435.513,A -85,B 0,C 180,E1 -23934.733,E2 -23934.733} C_VEL
LIN {X 0,Y 148.297,Z 429.423,A -85,B 0,C 180,E1 -23940.001,E2 -23940.001} C_VEL
LIN {X 0,Y 148.848,Z 421.803,A -85,B 0,C 180,E1 -23945.419,E2 -23945.419} C_VEL
LIN {X 0,Y 149.994,Z 412.473,A -85,B 0,C 180,E1 -23950.803,E2 -23950.803} C_VEL
LIN {X 0,Y 152.084,Z 401.351,A -85,B 0,C 180,E1 -23956.098,E2 -23956.098} C_VEL
LIN {X 0,Y 154.669,Z 389.677,A -85,B 0,C 180,E1 -23960.62,E2 -23960.62} C_VEL
LIN {X 0,Y 158.06,Z 375.84,A -85,B 0,C 180,E1 -23964.988,E2 -23964.988} C_VEL
LIN {X 0,Y 161.151,Z 363.098,A -85,B 0,C 180,E1 -23968.313,E2 -23968.313} C_VEL
LIN {X 0,Y 164.276,Z 349.798,A -85,B 0,C 180,E1 -23971.203,E2 -23971.203} C_VEL
LIN {X 0,Y 163.457,Z 344.548,A -85,B 0,C 180,E1 -23972.4,E2 -23972.4} C_VEL
LIN {X 0,Y 161.517,Z 336.296,A -85,B 0,C 180,E1 -23974.235,E2 -23974.235} C_VEL
LIN {X 0,Y 157.04,Z 321.167,A -85,B 0,C 180,E1 -23977.474,E2 -23977.474} C_VEL
LIN {X 0,Y 151.857,Z 306.309,A -85,B 0,C 180,E1 -23980.528,E2 -23980.528} C_VEL
LIN {X 0,Y 150.131,Z 301.418,A -85,B 0,C 180,E1 -23981.496,E2 -23981.496} C_VEL
LIN {X 0,Y 150.128,Z 301.412,A -85,B 0,C 180,E1 -23985.396,E2 -23985.396} C_VEL
LIN {X 0,Y 150.143,Z 301.408,A -85,B 0,C 180,E1 -23989.056,E2 -23989.056} C_VEL
LIN {X 0,Y 150.181,Z 301.403,A -85,B 0,C 180,E1 -23992.708,E2 -23992.708} C_VEL
LIN {X 0,Y 150.217,Z 301.398,A -85,B 0,C 180,E1 -23997.368,E2 -23997.368} C_VEL
LIN {X 0,Y 150.247,Z 301.395,A -85,B 0,C 180,E1 -24002.718,E2 -24002.718} C_VEL
LIN {X 0,Y 150.354,Z 301.38,A -85,B 0,C 180,E1 -24009.208,E2 -24009.208} C_VEL
LIN {X 0,Y 150.365,Z 301.377,A -85,B 0,C 180,E1 -24013.714,E2 -24013.714} C_VEL
LIN {X 0,Y 150.613,Z 301.348,A -85,B 0,C 180,E1 -24019.243,E2 -24019.243} C_VEL
LIN {X 0,Y 150.702,Z 301.335,A -85,B 0,C 180,E1 -24021.958,E2 -24021.958} C_VEL
LIN {X 0,Y 151.216,Z 301.27,A -85,B 0,C 180,E1 -24030,E2 -24030} C_VEL
LIN {X 0,Y 150.704,Z 301.334,A -85,B 0,C 180,E1 -24038.042,E2 -24038.042} C_VEL
LIN {X 0,Y 150.581,Z 301.35,A -85,B 0,C 180,E1 -24041.438,E2 -24041.438} C_VEL
LIN {X 0,Y 150.393,Z 301.373,A -85,B 0,C 180,E1 -24046.283,E2 -24046.283} C_VEL
LIN {X 0,Y 150.393,Z 301.375,A -85,B 0,C 180,E1 -24050.831,E2 -24050.831} C_VEL
LIN {X 0,Y 150.247,Z 301.391,A -85,B 0,C 180,E1 -24057.282,E2 -24057.282} C_VEL
LIN {X 0,Y 150.217,Z 301.396,A -85,B 0,C 180,E1 -24062.632,E2 -24062.632} C_VEL
LIN {X 0,Y 150.171,Z 301.404,A -85,B 0,C 180,E1 -24067.474,E2 -24067.474} C_VEL
LIN {X 0,Y 150.135,Z 301.404,A -85,B 0,C 180,E1 -24071.497,E2 -24071.497} C_VEL
LIN {X 0,Y 150.128,Z 301.409,A -85,B 0,C 180,E1 -24075.395,E2 -24075.395} C_VEL
LIN {X 0,Y 150.144,Z 301.405,A -85,B 0,C 180,E1 -24079.055,E2 -24079.055} C_VEL
LIN {X 0,Y 150.182,Z 301.401,A -85,B 0,C 180,E1 -24082.707,E2 -24082.707} C_VEL
LIN {X 0,Y 150.217,Z 301.395,A -85,B 0,C 180,E1 -24087.368,E2 -24087.368} C_VEL
LIN {X 0,Y 150.247,Z 301.396,A -85,B 0,C 180,E1 -24092.718,E2 -24092.718} C_VEL
LIN {X 0,Y 150.354,Z 301.379,A -85,B 0,C 180,E1 -24099.207,E2 -24099.207} C_VEL
LIN {X 0,Y 150.365,Z 301.378,A -85,B 0,C 180,E1 -24103.713,E2 -24103.713} C_VEL
LIN {X 0,Y 150.613,Z 301.348,A -85,B 0,C 180,E1 -24109.242,E2 -24109.242} C_VEL
LIN {X 0,Y 150.703,Z 301.336,A -85,B 0,C 180,E1 -24111.957,E2 -24111.957} C_VEL
LIN {X 0,Y 151.216,Z 301.272,A -85,B 0,C 180,E1 -24119.999,E2 -24119.999} C_VEL
LIN {X 0,Y 150.703,Z 301.336,A -85,B 0,C 180,E1 -24128.042,E2 -24128.042} C_VEL
LIN {X 0,Y 150.579,Z 301.349,A -85,B 0,C 180,E1 -24131.436,E2 -24131.436} C_VEL
LIN {X 0,Y 150.364,Z 301.377,A -85,B 0,C 180,E1 -24136.286,E2 -24136.286} C_VEL
LIN {X 0,Y 150.37,Z 301.381,A -85,B 0,C 180,E1 -24141.956,E2 -24141.956} C_VEL
LIN {X 0,Y 150.504,Z 301.457,A -85,B 0,C 180,E1 -24144.116,E2 -24144.116} C_VEL
LIN {X 0,Y 150.924,Z 305.575,A -85,B 0,C 180,E1 -24150.812,E2 -24150.812} C_VEL
LIN {X 0,Y 151.604,Z 308.523,A -85,B 0,C 180,E1 -24155.413,E2 -24155.413} C_VEL
LIN {X 0,Y 152.025,Z 310.432,A -85,B 0,C 180,E1 -24158.281,E2 -24158.281} C_VEL
LIN {X 0,Y 155.685,Z 322.52,A -85,B 0,C 180,E1 -24160.46,E2 -24160.46} C_VEL
LIN {X 0,Y 158.196,Z 331.549,A -85,B 0,C 180,E1 -24162.151,E2 -24162.151} C_VEL
LIN {X 0,Y 159.61,Z 340.454,A -85,B 0,C 180,E1 -24163.775,E2 -24163.775} C_VEL
LIN {X 0,Y 161.294,Z 354.354,A -85,B 0,C 180,E1 -24166.491,E2 -24166.491} C_VEL
LIN {X 0,Y 163.064,Z 369.982,A -85,B 0,C 180,E1 -24169.957,E2 -24169.957} C_VEL
LIN {X 0,Y 164.463,Z 383.178,A -85,B 0,C 180,E1 -24173.254,E2 -24173.254} C_VEL
LIN {X 0,Y 164.969,Z 387.555,A -85,B 0,C 180,E1 -24174.426,E2 -24174.426} C_VEL
LIN {X 0,Y 164.073,Z 391.242,A -85,B 0,C 180,E1 -24175.42,E2 -24175.42} C_VEL
LIN {X 0,Y 160.147,Z 403.091,A -85,B 0,C 180,E1 -24178.959,E2 -24178.959} C_VEL
LIN {X 0,Y 156.326,Z 414.869,A -85,B 0,C 180,E1 -24183.283,E2 -24183.283} C_VEL
LIN {X 0,Y 153.378,Z 424.783,A -85,B 0,C 180,E1 -24187.788,E2 -24187.788} C_VEL
LIN {X 0,Y 151.197,Z 433.13,A -85,B 0,C 180,E1 -24192.414,E2 -24192.414} C_VEL
LIN {X 0,Y 149.751,Z 441.033,A -85,B 0,C 180,E1 -24197.808,E2 -24197.808} C_VEL
LIN {X 0,Y 149.215,Z 446.693,A -85,B 0,C 180,E1 -24202.593,E2 -24202.593} C_VEL
LIN {X 0,Y 149.044,Z 451.066,A -85,B 0,C 180,E1 -24207.297,E2 -24207.297} C_VEL
LIN {X 0,Y 149.02,Z 453.088,A -85,B 0,C 180,E1 -24210,E2 -24210} C_VEL
LIN {X 0,Y 148.647,Z 456.094,A -85,B 0,C 180,E1 -24215.426,E2 -24215.426} C_VEL
LIN {X 0,Y 148.62,Z 457.951,A -85,B 0,C 180,E1 -24220.903,E2 -24220.903} C_VEL
LIN {X 0,Y 149.776,Z 459.028,A -85,B 0,C 180,E1 -24226.352,E2 -24226.352} C_VEL
LIN {X 0,Y 153.997,Z 459.21,A -85,B 0,C 180,E1 -24234.251,E2 -24234.251} C_VEL
LIN {X 0,Y 161.396,Z 457.929,A -85,B 0,C 180,E1 -24241.503,E2 -24241.503} C_VEL
LIN {X 0,Y 171.452,Z 455.333,A -85,B 0,C 180,E1 -24247.942,E2 -24247.942} C_VEL
LIN {X 0,Y 184.169,Z 451.58,A -85,B 0,C 180,E1 -24253.385,E2 -24253.385} C_VEL
LIN {X 0,Y 189.805,Z 449.807,A -85,B 0,C 180,E1 -24255.29,E2 -24255.29} C_VEL
LIN {X 0,Y 181.068,Z 450.93,A -85,B 0,C 180,E1 -24258.758,E2 -24258.758} C_VEL
LIN {X 0,Y 177.096,Z 451.366,A -85,B 0,C 180,E1 -24260.155,E2 -24260.155} C_VEL
LIN {X 0,Y 169.435,Z 451.968,A -85,B 0,C 180,E1 -24262.233,E2 -24262.233} C_VEL
LIN {X 0,Y 162.087,Z 452.049,A -85,B 0,C 180,E1 -24264.52,E2 -24264.52} C_VEL
LIN {X 0,Y 158.693,Z 451.739,A -85,B 0,C 180,E1 -24266.235,E2 -24266.235} C_VEL
LIN {X 0,Y 151.255,Z 449.948,A -85,B 0,C 180,E1 -24272.313,E2 -24272.313} C_VEL
LIN {X 0,Y 145.091,Z 446.077,A -85,B 0,C 180,E1 -24280.18,E2 -24280.18} C_VEL
LIN {X 0,Y 142.729,Z 442.397,A -85,B 0,C 180,E1 -24285.748,E2 -24285.748} C_VEL
LIN {X 0,Y 141.477,Z 437.691,A -85,B 0,C 180,E1 -24291.43,E2 -24291.43} C_VEL
LIN {X 0,Y 141.171,Z 431.899,A -85,B 0,C 180,E1 -24297.147,E2 -24297.147} C_VEL
LIN {X 0,Y 141.314,Z 426.659,A -85,B 0,C 180,E1 -24301.426,E2 -24301.426} C_VEL
LIN {X 0,Y 141.937,Z 419.496,A -85,B 0,C 180,E1 -24306.397,E2 -24306.397} C_VEL
LIN {X 0,Y 143.061,Z 411.059,A -85,B 0,C 180,E1 -24311.333,E2 -24311.333} C_VEL
LIN {X 0,Y 145.315,Z 399.508,A -85,B 0,C 180,E1 -24316.87,E2 -24316.87} C_VEL
LIN {X 0,Y 148.04,Z 387.549,A -85,B 0,C 180,E1 -24321.588,E2 -24321.588} C_VEL
LIN {X 0,Y 151.363,Z 374.467,A -85,B 0,C 180,E1 -24325.805,E2 -24325.805} C_VEL
LIN {X 0,Y 154.575,Z 361.421,A -85,B 0,C 180,E1 -24329.26,E2 -24329.26} C_VEL
LIN {X 0,Y 157.291,Z 349.556,A -85,B 0,C 180,E1 -24331.902,E2 -24331.902} C_VEL
LIN {X 0,Y 154.798,Z 338.308,A -85,B 0,C 180,E1 -24334.598,E2 -24334.598} C_VEL
LIN {X 0,Y 150.522,Z 323.706,A -85,B 0,C 180,E1 -24337.939,E2 -24337.939} C_VEL
LIN {X 0,Y 145.655,Z 309.474,A -85,B 0,C 180,E1 -24341.069,E2 -24341.069} C_VEL
LIN {X 0,Y 143.088,Z 302.292,A -85,B 0,C 180,E1 -24342.646,E2 -24342.646} C_VEL
LIN {X 0,Y 143.042,Z 302.29,A -85,B 0,C 180,E1 -24347.477,E2 -24347.477} C_VEL
LIN {X 0,Y 143.077,Z 302.287,A -85,B 0,C 180,E1 -24351.807,E2 -24351.807} C_VEL
LIN {X 0,Y 143.184,Z 302.274,A -85,B 0,C 180,E1 -24357.322,E2 -24357.322} C_VEL
LIN {X 0,Y 143.193,Z 302.273,A -85,B 0,C 180,E1 -24362.063,E2 -24362.063} C_VEL
LIN {X 0,Y 143.28,Z 302.262,A -85,B 0,C 180,E1 -24368.746,E2 -24368.746} C_VEL
LIN {X 0,Y 143.304,Z 302.256,A -85,B 0,C 180,E1 -24372.887,E2 -24372.887} C_VEL
LIN {X 0,Y 143.539,Z 302.23,A -85,B 0,C 180,E1 -24378.706,E2 -24378.706} C_VEL
LIN {X 0,Y 143.624,Z 302.217,A -85,B 0,C 180,E1 -24381.559,E2 -24381.559} C_VEL
LIN {X 0,Y 144.175,Z 302.147,A -85,B 0,C 180,E1 -24390,E2 -24390} C_VEL
LIN {X 0,Y 143.626,Z 302.215,A -85,B 0,C 180,E1 -24398.442,E2 -24398.442} C_VEL
LIN {X 0,Y 143.51,Z 302.232,A -85,B 0,C 180,E1 -24401.634,E2 -24401.634} C_VEL
LIN {X 0,Y 143.334,Z 302.252,A -85,B 0,C 180,E1 -24407.109,E2 -24407.109} C_VEL
LIN {X 0,Y 143.314,Z 302.258,A -85,B 0,C 180,E1 -24411.29,E2 -24411.29} C_VEL
LIN {X 0,Y 143.193,Z 302.272,A -85,B 0,C 180,E1 -24417.937,E2 -24417.937} C_VEL
LIN {X 0,Y 143.145,Z 302.274,A -85,B 0,C 180,E1 -24423.419,E2 -24423.419} C_VEL
LIN {X 0,Y 143.054,Z 302.289,A -85,B 0,C 180,E1 -24429.693,E2 -24429.693} C_VEL
LIN {X 0,Y 143.035,Z 302.29,A -85,B 0,C 180,E1 -24433.464,E2 -24433.464} C_VEL
LIN {X 0,Y 143.042,Z 302.291,A -85,B 0,C 180,E1 -24437.476,E2 -24437.476} C_VEL
LIN {X 0,Y 143.078,Z 302.283,A -85,B 0,C 180,E1 -24441.807,E2 -24441.807} C_VEL
LIN {X 0,Y 143.184,Z 302.271,A -85,B 0,C 180,E1 -24447.321,E2 -24447.321} C_VEL
LIN {X 0,Y 143.193,Z 302.272,A -85,B 0,C 180,E1 -24452.063,E2 -24452.063} C_VEL
LIN {X 0,Y 143.28,Z 302.26,A -85,B 0,C 180,E1 -24458.745,E2 -24458.745} C_VEL
LIN {X 0,Y 143.305,Z 302.258,A -85,B 0,C 180,E1 -24462.886,E2 -24462.886} C_VEL
LIN {X 0,Y 143.539,Z 302.23,A -85,B 0,C 180,E1 -24468.705,E2 -24468.705} C_VEL
LIN {X 0,Y 143.625,Z 302.218,A -85,B 0,C 180,E1 -24471.558,E2 -24471.558} C_VEL
LIN {X 0,Y 144.175,Z 302.149,A -85,B 0,C 180,E1 -24479.999,E2 -24479.999} C_VEL
LIN {X 0,Y 143.625,Z 302.216,A -85,B 0,C 180,E1 -24488.441,E2 -24488.441} C_VEL
LIN {X 0,Y 143.507,Z 302.231,A -85,B 0,C 180,E1 -24491.629,E2 -24491.629} C_VEL
LIN {X 0,Y 143.307,Z 302.257,A -85,B 0,C 180,E1 -24497.112,E2 -24497.112} C_VEL
LIN {X 0,Y 143.385,Z 302.252,A -85,B 0,C 180,E1 -24503.086,E2 -24503.086} C_VEL
LIN {X 0,Y 143.489,Z 302.538,A -85,B 0,C 180,E1 -24504.602,E2 -24504.602} C_VEL
LIN {X 0,Y 143.686,Z 305.293,A -85,B 0,C 180,E1 -24509.282,E2 -24509.282} C_VEL
LIN {X 0,Y 144.55,Z 309.206,A -85,B 0,C 180,E1 -24515.692,E2 -24515.692} C_VEL
LIN {X 0,Y 144.727,Z 310.016,A -85,B 0,C 180,E1 -24516.936,E2 -24516.936} C_VEL
LIN {X 0,Y 150.251,Z 328.224,A -85,B 0,C 180,E1 -24520.486,E2 -24520.486} C_VEL
LIN {X 0,Y 152.519,Z 338.502,A -85,B 0,C 180,E1 -24522.5,E2 -24522.5} C_VEL
LIN {X 0,Y 154.339,Z 354.726,A -85,B 0,C 180,E1 -24525.822,E2 -24525.822} C_VEL
LIN {X 0,Y 155.849,Z 368.695,A -85,B 0,C 180,E1 -24529.053,E2 -24529.053} C_VEL
LIN {X 0,Y 157.228,Z 381.755,A -85,B 0,C 180,E1 -24532.436,E2 -24532.436} C_VEL
LIN {X 0,Y 157.82,Z 387.478,A -85,B 0,C 180,E1 -24534.049,E2 -24534.049} C_VEL
LIN {X 0,Y 157.218,Z 390.344,A -85,B 0,C 180,E1 -24534.862,E2 -24534.862} C_VEL
LIN {X 0,Y 152.888,Z 403.086,A -85,B 0,C 180,E1 -24538.859,E2 -24538.859} C_VEL
LIN {X 0,Y 149.102,Z 414.639,A -85,B 0,C 180,E1 -24543.364,E2 -24543.364} C_VEL
LIN {X 0,Y 146.134,Z 424.496,A -85,B 0,C 180,E1 -24548.116,E2 -24548.116} C_VEL
LIN {X 0,Y 143.841,Z 433.833,A -85,B 0,C 180,E1 -24553.683,E2 -24553.683} C_VEL
LIN {X 0,Y 142.682,Z 440.526,A -85,B 0,C 180,E1 -24558.637,E2 -24558.637} C_VEL
LIN {X 0,Y 142.301,Z 445.37,A -85,B 0,C 180,E1 -24562.907,E2 -24562.907} C_VEL
LIN {X 0,Y 142.152,Z 449.247,A -85,B 0,C 180,E1 -24567.166,E2 -24567.166} C_VEL
LIN {X 0,Y 142.125,Z 451.417,A -85,B 0,C 180,E1 -24570,E2 -24570} C_VEL
LIN {X 0,Y 141.879,Z 453.153,A -85,B 0,C 180,E1 -24572.839,E2 -24572.839} C_VEL
LIN {X 0,Y 141.624,Z 455.167,A -85,B 0,C 180,E1 -24577.032,E2 -24577.032} C_VEL
LIN {X 0,Y 142.188,Z 457.362,A -85,B 0,C 180,E1 -24584.308,E2 -24584.308} C_VEL
LIN {X 0,Y 145.634,Z 458.397,A -85,B 0,C 180,E1 -24592.71,E2 -24592.71} C_VEL
LIN {X 0,Y 152.464,Z 457.977,A -85,B 0,C 180,E1 -24600.468,E2 -24600.468} C_VEL
LIN {X 0,Y 162.099,Z 456.236,A -85,B 0,C 180,E1 -24607.372,E2 -24607.372} C_VEL
LIN {X 0,Y 170.026,Z 454.425,A -85,B 0,C 180,E1 -24611.404,E2 -24611.404} C_VEL
LIN {X 0,Y 180.464,Z 451.771,A -85,B 0,C 180,E1 -24615.494,E2 -24615.494} C_VEL
LIN {X 0,Y 167.584,Z 452.383,A -85,B 0,C 180,E1 -24621.02,E2 -24621.02} C_VEL
LIN {X 0,Y 158.693,Z 451.739,A -85,B 0,C 180,E1 -24626.235,E2 -24626.235} C_VEL
LIN {X 0,Y 155.47,Z 451.344,A -85,B 0,C 180,E1 -24628.032,E2 -24628.032} C_VEL
LIN {X 0,Y 149.001,Z 450.341,A -85,B 0,C 180,E1 -24630.829,E2 -24630.829} C_VEL
LIN {X 0,Y 142.998,Z 448.802,A -85,B 0,C 180,E1 -24633.862,E2 -24633.862} C_VEL
LIN {X 0,Y 140.598,Z 447.636,A -85,B 0,C 180,E1 -24635.993,E2 -24635.993} C_VEL
LIN {X 0,Y 136.372,Z 442.975,A -85,B 0,C 180,E1 -24643.535,E2 -24643.535} C_VEL
LIN {X 0,Y 134.723,Z 438.317,A -85,B 0,C 180,E1 -24649.481,E2 -24649.481} C_VEL
LIN {X 0,Y 134.165,Z 431.966,A -85,B 0,C 180,E1 -24656.073,E2 -24656.073} C_VEL
LIN {X 0,Y 134.289,Z 425.602,A -85,B 0,C 180,E1 -24661.5,E2 -24661.5} C_VEL
LIN {X 0,Y 134.822,Z 419.297,A -85,B 0,C 180,E1 -24665.985,E2 -24665.985} C_VEL
LIN {X 0,Y 136.161,Z 409.434,A -85,B 0,C 180,E1 -24671.916,E2 -24671.916} C_VEL
LIN {X 0,Y 138.22,Z 399.226,A -85,B 0,C 180,E1 -24677,E2 -24677} C_VEL
LIN {X 0,Y 141.005,Z 387.132,A -85,B 0,C 180,E1 -24681.952,E2 -24681.952} C_VEL
LIN {X 0,Y 144.424,Z 374.026,A -85,B 0,C 180,E1 -24686.363,E2 -24686.363} C_VEL
LIN {X 0,Y 147.76,Z 361.026,A -85,B 0,C 180,E1 -24689.962,E2 -24689.962} C_VEL
LIN {X 0,Y 150.238,Z 351.057,A -85,B 0,C 180,E1 -24692.264,E2 -24692.264} C_VEL
LIN {X 0,Y 148.808,Z 343.127,A -85,B 0,C 180,E1 -24694.261,E2 -24694.261} C_VEL
LIN {X 0,Y 145.101,Z 329.907,A -85,B 0,C 180,E1 -24697.521,E2 -24697.521} C_VEL
LIN {X 0,Y 141.109,Z 317.328,A -85,B 0,C 180,E1 -24700.468,E2 -24700.468} C_VEL
LIN {X 0,Y 136.028,Z 303.169,A -85,B 0,C 180,E1 -24703.764,E2 -24703.764} C_VEL
LIN {X 0,Y 135.986,Z 303.169,A -85,B 0,C 180,E1 -24707.789,E2 -24707.789} C_VEL
LIN {X 0,Y 136.027,Z 303.166,A -85,B 0,C 180,E1 -24711.684,E2 -24711.684} C_VEL
LIN {X 0,Y 136.087,Z 303.158,A -85,B 0,C 180,E1 -24715.721,E2 -24715.721} C_VEL
LIN {X 0,Y 136.149,Z 303.151,A -85,B 0,C 180,E1 -24722.317,E2 -24722.317} C_VEL
LIN {X 0,Y 136.247,Z 303.138,A -85,B 0,C 180,E1 -24728.833,E2 -24728.833} C_VEL
LIN {X 0,Y 136.271,Z 303.13,A -85,B 0,C 180,E1 -24735.056,E2 -24735.056} C_VEL
LIN {X 0,Y 136.434,Z 303.115,A -85,B 0,C 180,E1 -24738.165,E2 -24738.165} C_VEL
LIN {X 0,Y 136.551,Z 303.098,A -85,B 0,C 180,E1 -24741.118,E2 -24741.118} C_VEL
LIN {X 0,Y 137.132,Z 303.024,A -85,B 0,C 180,E1 -24750,E2 -24750} C_VEL
LIN {X 0,Y 136.552,Z 303.095,A -85,B 0,C 180,E1 -24758.882,E2 -24758.882} C_VEL
LIN {X 0,Y 136.461,Z 303.111,A -85,B 0,C 180,E1 -24761.889,E2 -24761.889} C_VEL
LIN {X 0,Y 136.274,Z 303.13,A -85,B 0,C 180,E1 -24768.025,E2 -24768.025} C_VEL
LIN {X 0,Y 136.23,Z 303.141,A -85,B 0,C 180,E1 -24771.78,E2 -24771.78} C_VEL
LIN {X 0,Y 136.103,Z 303.155,A -85,B 0,C 180,E1 -24778.616,E2 -24778.616} C_VEL
LIN {X 0,Y 136.044,Z 303.157,A -85,B 0,C 180,E1 -24784.629,E2 -24784.629} C_VEL
LIN {X 0,Y 136.027,Z 303.166,A -85,B 0,C 180,E1 -24789.194,E2 -24789.194} C_VEL
LIN {X 0,Y 135.98,Z 303.169,A -85,B 0,C 180,E1 -24793.648,E2 -24793.648} C_VEL
LIN {X 0,Y 135.986,Z 303.17,A -85,B 0,C 180,E1 -24797.788,E2 -24797.788} C_VEL
LIN {X 0,Y 136.027,Z 303.162,A -85,B 0,C 180,E1 -24801.683,E2 -24801.683} C_VEL
LIN {X 0,Y 136.087,Z 303.157,A -85,B 0,C 180,E1 -24805.721,E2 -24805.721} C_VEL
LIN {X 0,Y 136.149,Z 303.15,A -85,B 0,C 180,E1 -24812.316,E2 -24812.316} C_VEL
